// TwinCAT 3 PLC project ProgramPLC
// ProgramVersion: 3.1.4026.19
// libraries:
//   Tc2_DataExchange, * (Beckhoff Automation GmbH)
//   Tc2_Drive, * (Beckhoff Automation GmbH)
//   Tc2_EtherCAT, * (Beckhoff Automation GmbH)
//   Tc2_IoFunctions, * (Beckhoff Automation GmbH)
//   Tc2_Math, * (Beckhoff Automation GmbH)
//   Tc2_MC2, * (Beckhoff Automation GmbH)
//   Tc2_MC2_Camming, * (Beckhoff Automation GmbH)
//   Tc2_MC2_Drive, * (Beckhoff Automation GmbH)
//   Tc2_MC2_FlyingSaw, * (Beckhoff Automation GmbH)
//   Tc2_NC, * (Beckhoff Automation GmbH)
//   Tc2_Standard, * (Beckhoff Automation GmbH)
//   Tc2_SUPS, * (Beckhoff Automation GmbH)
//   Tc2_System, * (Beckhoff Automation GmbH)
//   Tc2_Utilities, * (Beckhoff Automation GmbH)
//   Tc3_EventLogger, * (Beckhoff Automation GmbH)
//   Tc3_Interfaces, * (Beckhoff Automation GmbH)
//   Tc3_IoLink, * (Beckhoff Automation GmbH)
//   Tc3_MC2_AdvancedHoming, * (Beckhoff Automation GmbH)
//   Tc3_Module, * (Beckhoff Automation GmbH)
//   Tc3_PackML, * (Beckhoff Automation GmbH)
//   TcEventLogger, * (Beckhoff Automation Poland)
//   Festo_VTEM_DevCon,3.5.7.235,Festo SE & Co. KG
// project tree:
//   DUTs/AxisControl/ ST_AxisControlHoldingBrake.TcDUT, ST_AxisControlLS.TcDUT, ST_AxisControlManual.TcDUT, ST_AxisControlManualHMI.TcDUT
//   DUTs/CapPreScrewer/ E_CapPreScrewer.TcDUT, ST_ADS_Read_Write.TcDUT, ST_ADS_Write.TcDUT, ST_CapPreScrewerCommandsIn.TcDUT, ST_CapPreScrewerParameters.TcDUT, ST_FormsCapSorter.TcDUT
//   DUTs/DUTsAdsCommunication/ ST_Communication.TcDUT, ST_MachinePermissions.TcDUT, ST_PackMLCmdForCom.TcDUT, ST_ReservedSignals.TcDUT
//   DUTs/DUTsAxisOnline/FBsIO/ ST_FBGetDriveRefIO.TcDUT, ST_FBHoldingBrakeCtrlIO.TcDUT, ST_FBMotorMonitoringIO.TcDUT, ST_FBNcSWLimitSwitchCtrlIO.TcDUT, ST_FBReadChannelErrorCodeIO.TcDUT, ST_FBSetPositionOffsetIO.TcDUT, ST_McAxisOnlineErrorCollection.TcDUT, ST_McAxisStatus.TcDUT, ST_MCHaltIO.TcDUT, ST_MCHomeIO.TcDUT, ST_MCJogIO.TcDUT, ST_MCMoveAbsoluteIO.TcDUT, ST_MCMoveModuloIO.TcDUT, ST_MCMoveRelativeIO.TcDUT, ST_MCMoveVelocityIO.TcDUT, ST_MCPowerIO.TcDUT, ST_MCReadDriveAddressIO.TcDUT, ST_MCReadParameterSetIO.TcDUT, ST_MCResetIO.TcDUT, ST_MCSetPositionIO.TcDUT, ST_MCStopIO.TcDUT
//   DUTs/DUTsAxisOnline/ ST_AX5000Diag.TcDUT, ST_McAxisOnline.TcDUT
//   DUTs/DUTsDiagnostics/ E_DiagState.TcDUT, ST_FrmWcDiag.TcDUT
//   DUTs/DUTsNew/ E_Actuator.TcDUT, E_Barrier.TcDUT, E_WeightLiftStationState.TcDUT
//   DUTs/DUTsPackMLStateMachine/ E_PackMLCommand.TcDUT, E_PackMLMode.TcDUT, E_PackMLState.TcDUT
//   DUTs/ E_BottleFeederState.TcDUT, E_CapFeederState.TcDUT, E_CapFeederState_1.TcDUT, E_CapPushingState.TcDUT, E_CatchStationState.TcDUT, E_CheckerState.TcDUT, E_ConveyorState.TcDUT, E_DispencerLifterState.TcDUT, E_DispencerState.TcDUT, E_DragStationState.TcDUT, E_DragStationStatePneum.TcDUT, E_EntranceGatesState.TcDUT, E_FestoEmcsStState.TcDUT, E_GripperScrewer.TcDUT, E_MachineState.TcDUT, E_MassHeatingState.TcDUT, E_PuckInserterState.TcDUT, E_RobotMovState.TcDUT, E_RollerScrewer.TcDUT, E_Station.TcDUT, E_WeightState.TcDUT, ST_MoverState.TcDUT, ST_Point.TcDUT, ST_Point_1.TcDUT, ST_SlotStatus.TcDUT, S_CycleTimes.TcDUT, S_Error.TcDUT, S_Information.TcDUT, S_PackageState.TcDUT, S_RFIDCheck.TcDUT, S_Warning.TcDUT
//   DUTs/ServerClientENUMS/ E_ConnectionSteps.TcDUT, E_ServerSteps.TcDUT
//   DUTs/Stations/LidFeeder/ E_LidFeederState.TcDUT
//   DUTs/Stations/LidSealer/ E_LidSealing.TcDUT
//   DUTs/Stations/WickFeeder/ E_WickFeederSorterState.TcDUT, E_WickFeederState.TcDUT
//   / GlobalTextList.TcGTLO, PlcTask.TcTTO, WeightTask.TcTTO
//   GVLs/ GVL.TcGVL, gvlChecks.TcGVL, gvlCommunication.TcGVL, GVL_CP.TcGVL, GVL_IO.TcGVL, GVL_ROPP.TcGVL, GVL_RS.TcGVL, Iterators.TcGVL, VIS.TcGVL, VIS_CP.TcGVL, VIS_M.TcGVL, VIS_RFID.TcGVL, VIS_ROPP.TcGVL, VIS_RS.TcGVL
//   GVLs/UVFF/ GVL_Recipe.TcGVL, GVL_UVFF.TcGVL, GVL_VIS.TcGVL
//   POUs/FB/ADSCommumication/ FB_AdsCommunicationRead.TcPOU
//   POUs/FB/AxisControl/AX8000/ FB_AxisAX8000.TcPOU, I_AxisControlPhysical.TcIO
//   POUs/FB/AxisControl/Base/ FB_AxisBase.TcPOU, I_AxisControlBase.TcIO
//   POUs/FB/AxisControl/Internal/ FB_FilterEx_2.TcPOU, FB_GetDriveRef_1.TcPOU, FB_HoldingBrakeCtrlAX8000_1.TcPOU, FB_NcPosLagMonitoring.TcPOU, FB_NcSWLimitSwitchCtrlv2.TcPOU, FB_ReadChannelErrorCodeAX8000_1.TcPOU, F_AX8xErrMsg_2.TcPOU, F_AxErrMsg_2.TcPOU
//   POUs/FB/AxisControl/Internal/HomingAdv/ FB_HomingLimitSwitch.TcPOU, FB_HomingMemoryAX8000.TcPOU, FB_HomingTorqueDetection.TcPOU, FB_HomingTorqueDetectionSensor.TcPOU, FB_HomingTorque_1.TcPOU
//   POUs/FB/Axis/ F_AX8xErrMsg.TcPOU, F_AxErrMsg.TcPOU
//   POUs/FB/Blinkers/ FB_Blink_AS.TcPOU, FB_Blink_S.TcPOU, FUN_Beep.TcPOU
//   POUs/FB/Charts/ FB_ChartGenerator.TcPOU, FB_SimplePulseGenerator.TcPOU, FB_WeightHistory.TcPOU
//   POUs/FB/Conversions/ ArrayOfReal_To_String.TcPOU, arrBOOL16_TO_WORD.TcPOU, arrBOOL8_TO_BYTE.TcPOU, ArrOfInt_To_String.TcPOU, FB_CONCAT_S2040.TcPOU, FB_DIntTo4Byte.TcPOU, FB_IntTo2Byte.TcPOU, F_4BYTES_TO_DWORD.TcPOU, F_4BYTES_TO_REAL.TcPOU, F_8BYTES_TO_LREAL.TcPOU, F_BCDToDec.TcPOU, F_CLEAN_S2040.TcPOU, F_Convert_4BBCD_To_Real.TcPOU, F_DWORD_TO_REAL.TcPOU, F_Words_to_Real.TcPOU, GRAYB_TO_WORD.TcPOU, GRAYW_TO_WORD.TcPOU
//   POUs/FB/Conversions/BitOriented/ BCD_TO_INT.TcPOU, F_1stByteW.TcPOU, F_1stByteWtoB.TcPOU, F_2Bytes_To_Word.TcPOU, F_2ndByteW.TcPOU, F_2ndByteWtoB.TcPOU, F_MaskWord.TcPOU, L_TBConvArrBitsToDword.TcPOU, L_TBConvBitsToByte.TcPOU, L_TBConvBitsToDword.TcPOU, L_TBConvBitsToWord.TcPOU, L_TBConvByteToBits.TcPOU, L_TBConvDwordToArrBits.TcPOU, L_TBConvDwordToBits.TcPOU, L_TBConvWordToBits.TcPOU, L_TBGetBitOfByte.TcPOU, L_TBGetBitOfDword.TcPOU, L_TBGetBitOfWord.TcPOU, L_TBResetBitOfByte.TcPOU, L_TBResetBitOfDword.TcPOU, L_TBResetBitOfWord.TcPOU, L_TBSetBitOfByte.TcPOU, L_TBSetBitOfDword.TcPOU, L_TBSetBitOfWord.TcPOU, L_TBSquareWave.TcPOU
//   POUs/FB/DateAndTime/ FB_GetSystemTime.TcPOU, FB_SimpleWorkTime.TcPOU, FB_TimeMeasureEx.TcPOU, FB_WorktimeCompact.TcPOU
//   POUs/FB/Diagnostics/FBsDiagnostic/ FB_AdvancedLogEvent.TcPOU, FB_AntiBlinkAlarmFilter.TcPOU, FB_TaskInfo.TcPOU
//   POUs/FB/Diagnostics/POUsDiagnosticComponents/Checks/ CheckBounds.TcPOU, CheckDivDInt.TcPOU, CheckDivLInt.TcPOU, CheckDivLReal.TcPOU, CheckDivReal.TcPOU, CheckPointer.TcPOU, CheckRangeSigned.TcPOU, CheckRangeUnsigned.TcPOU, P_Checks.TcPOU
//   POUs/FB/Diagnostics/POUsDiagnosticComponents/ P_EtherCAT_ChangeCounter.TcPOU, P_EtherCAT_Diag.TcPOU, P_GroupsWcStates.TcPOU, P_Persistent.TcPOU, P_PlcTaskSystemInfo.TcPOU, P_SystemDiag_EventLog.TcPOU, P_SystemInfo.TcPOU, P_TaskInfo.TcPOU
//   POUs/FB/ FB_2GripperScrewers.TcPOU, FB_2GripperScrewers_New.TcPOU, FB_2ReasonBadPackageWithID.TcPOU, FB_BalluffBMP0005.TcPOU, FB_BeckhoffEL3356Weight.TcPOU, FB_CapFeeder.TcPOU, FB_CapPreScrewer.TcPOU, FB_CapPusher.TcPOU, FB_CapPusherFeeder.TcPOU, FB_DigitalInput_1.TcPOU, FB_Robot2Bottles.TcPOU, FB_CapFeeder_old.TcPOU, FB_CatchStation.TcPOU, FB_CatchStationEnkoder.TcPOU, FB_CatchStationEnkoder_old.TcPOU (excluded from build), FB_Checker.TcPOU, FB_CycleTimes.TcPOU, FB_EntranceGatesServo.TcPOU, FB_FestoEmcsSt.TcPOU, FB_HomingTorque.TcPOU, FB_IfmIoLinkRfid.TcPOU, FB_InputFilter.TcPOU, FB_JiesangActuatorEncoder.TcPOU, FB_JiesangActuatorEncoder_1.TcPOU, FB_JiesangActuatorEncoderModul.TcPOU, FB_LenzeInverter.TcPOU, FB_LidFeeder.TcPOU, FB_LidSealer.TcPOU, FB_MitsubishiInverter.TcPOU, FB_MoveRegister.TcPOU, FB_MoveRegister4.TcPOU, FB_MoveRegisterCapControl.TcPOU, FB_MoveRegisterROPPCapControl.TcPOU, FB_MoveRegisterSortAndMove.TcPOU, FB_MoveRegisterSortAndMoveLF.TcPOU, FB_MoveRegisterLF.TcPOU, FB_MoveRegisterSortAndMoveROPP.TcPOU, FB_OEECycleTimes.TcPOU, FB_OEERejectionReason.TcPOU, FB_ReasonBadPackage.TcPOU, FB_RollerScrewer.TcPOU, FB_ROPPCapping.TcPOU, FB_ROPPFeeder.TcPOU, FB_SensorDiag.TcPOU, FB_ServoDispencerServoLifter.TcPOU, FB_ServoDispencerServoLifter_kopia_przed_akt_XTS.TcPOU, FB_SpringGateV2.TcPOU, FB_State.TcPOU, FB_TankHeating.TcPOU, FB_TempRegulator.TcPOU, FB_VisionChecker.TcPOU, FB_VisionChecker_new.TcPOU, FB_WeightCorrection.TcPOU, FB_WickFeederStation.TcPOU, FB_WriteDataToArrayOfArrays.TcPOU, FB_WriteDataToArrayString.TcPOU, FB_WriteRFID.TcPOU, FB_WriteRFIDnew.TcPOU, FB_AutoTrialRenew_ADS.TcPOU, F_StringToWstringPL.TcPOU, FB_InputFilter_v2.TcPOU
//   POUs/FB/FileAccess/ FB_ReadTextFromFile.TcPOU, FB_SaveTextToFile.TcPOU, FB_FileLog.TcPOU, FB_SaveLineToFile.TcPOU
//   POUs/FB/Led/ FB_PackMlToRgb_EL2564.TcPOU, FB_RgbLedTape_EL2563.TcPOU
//   POUs/FB/NC/ FB_PWM_BASIC.TcPOU
//   POUs/FB/NewFBs/ FB_BottleFeeder.TcPOU, FB_CatchStationWithSensor.TcPOU, FB_FormsDragStepper.TcPOU, FB_FormsDragActuator.TcPOU, FB_Gate.TcPOU, FB_PucksInserter.TcPOU, FB_SensorAcetone.TcPOU, FB_SensorFlow.TcPOU, FB_WeightStation.TcPOU
//   POUs/FB/POUsAxisOnline/AX5000/ FB_AxisDiag.TcPOU, FB_ChangeEtherCATSlaveState.TcPOU, FB_HoldingBrakeCtrlAX5000.TcPOU, FB_McAxisOnlineAX5000.TcPOU, FB_MotorMonitoringAX5000.TcPOU, FB_SetPositionOffset.TcPOU, F_AX5xErrMsg.TcPOU
//   POUs/FB/POUsAxisOnline/AX8000/ FB_HoldingBrakeCtrlAX8000.TcPOU, FB_McAxisOnlineAX8000.TcPOU, FB_MotorMonitoringAX8000.TcPOU, FB_ReadChannelErrorCodeAX8000.TcPOU, F_AX8xErrMsg_1.TcPOU
//   POUs/FB/POUsAxisOnline/EL72xx/ FB_HoldingBrakeCtrlEL72xx.TcPOU, FB_McAxisOnlineEL72xx.TcPOU, FB_MotorMonitoringEL72xx.TcPOU, FB_ReadChannelErrorCodeEL72xx.TcPOU, F_EL72ErrMsg.TcPOU
//   POUs/FB/POUsAxisOnline/FBs/ FB_FilterEx_1.TcPOU, FB_GetDriveRef.TcPOU, FB_NcSWLimitSwitchCtrl.TcPOU, F_AxErrMsg_1.TcPOU
//   POUs/FB/POUsAxisOnline/NC/ FB_McAxisOnlineNC.TcPOU
//   POUs/FB/Various/ FB_4_20mA_TO_INT.TcPOU, FB_Average.TcPOU, FB_FilterEx.TcPOU, FB_Persistent.TcPOU, FB_PIDBasic.TcPOU, FB_Skalowanie.TcPOU, F_ScaleLREAL.TcPOU, F_Scaling.TcPOU
//   POUs/ MAIN.TcPOU, P00_Alarms.TcPOU, P00_Basic.TcPOU, P00_Counters.TcPOU, P00_OEE.TcPOU, P00_Persistent.TcPOU, P00_Communication.TcPOU, P00_PneumaticValves.TcPOU, P00_ReadRFIDCard.TcPOU, P00_Recipes.TcPOU, P00_SensorDiagnostics.TcPOU, P00_Signalization.TcPOU, P00_SystemDiagnostics.TcPOU, P00_Visualization.TcPOU, P01_BottleFeeder.TcPOU, P00_PackML.TcPOU, P01_BottleSorter.TcPOU, P01_PucksInserter.TcPOU, P01_TwoPhasesBarriers.TcPOU, P02_BottlePusher.TcPOU, P02_Dispencers.TcPOU, P05_Weight.TcPOU, P06_WickFeeder.TcPOU, P07_CapPusher.TcPOU, P07_ROPP.TcPOU, P08_CapFeeder.TcPOU, P01_Gates.TcPOU, P05_WeightCorrection.TcPOU, P06_LidFeeder.TcPOU, P06_LidPuttedCheck.TcPOU, P06_LidSealer.TcPOU, P08_CapSorter.TcPOU, P09_CapPuttedCheck.TcPOU, P10_GripperScrewer.TcPOU, P11_CapCorrectCheck.TcPOU, P11_RollerScrewer.TcPOU, P13_BottleTransferAfterDrag.TcPOU, P13_BottleTransfer.TcPOU, P14_BadBottleConyevor.TcPOU, P15_FormTransporters.TcPOU, P16_LabelMachine.TcPOU, P17_TurnTables.TcPOU, P02_DispencersCharts.TcPOU, P200_CapPreScrewer.TcPOU, P20_ExhaustFan.TcPOU, P20_ExhaustFan_old.TcPOU, P_AdsLicenseServer.TcPOU, P_WenglorTeach.TcPOU
//   POUs/Recipes/NewRecipes/Components/ ST_BoolParametr.TcDUT, ST_DiParametrr.TcDUT, ST_LrParametr.TcDUT, ST_TextListParametr.TcDUT, ST_UdiParametr.TcDUT
//   POUs/Recipes/NewRecipes/ E_MacroProductProcessRegister.TcDUT, E_ProductType.TcDUT, ST_Recipe.TcDUT, ST_RecipeListItem.TcDUT, ST_Recipe_UBF_PARAM.TcDUT, ST_Recipe_UBL_PARAM.TcDUT, ST_Recipe_UCF_PARAM.TcDUT
//   POUs/Recipes/NewRecipes/RecipeCSV/ FB_ListSaveCSV.TcPOU, FB_LoadCSV.TcPOU, FB_RecipeSaveCSV.TcPOU, FB_RecipeVariablesSaveCSV.TcPOU
//   POUs/Recipes/NewRecipes/RecipeList/ E_FileOpSteps.TcDUT, FB_Load.TcPOU, FB_Save.TcPOU
//   POUs/Recipes/NewRecipes/RecipeParts/ ST_BoxRobotRecipe.TcDUT, ST_DownTransporterRecipe.TcDUT, ST_DymmyStationRecipe.TcDUT, ST_ExtMachineRecipe.TcDUT, ST_InBoxControlRecipe.TcDUT, ST_InTransporterRecipe.TcDUT, ST_LeftRightCloserValveRecipe.TcDUT, ST_LiftedTableRecipe.TcDUT, ST_LRTransporterRecipe.TcDUT, ST_MacroBoxFeedingProcessRecipe.TcDUT, ST_MacroBoxingProcessRecipe.TcDUT, ST_MacroInProcessRecipe.TcDUT, ST_MacroMachineProcessRecipe.TcDUT, ST_MacroProductProcessRecipe.TcDUT, ST_MacroTransportRecipe.TcDUT, ST_MainProcessRecipe.TcDUT, ST_MainSystemRecipe.TcDUT, ST_MoverPressValveRecipe.TcDUT, ST_OutControlRecipe.TcDUT, ST_ProductBoxerRecipe.TcDUT, ST_ProductRobotRecipe.TcDUT, ST_ProductTableCoverRecipe.TcDUT, ST_RejectBuforRecipe.TcDUT, ST_SpareElementsLockRecipe.TcDUT, ST_StandartGateRecipe.TcDUT, ST_StepMoverRecipe.TcDUT
//   POUs/Recipes/ P009_ReadSavePersistent.TcPOU, P010_AlarmsWarningsInfosLogs.TcPOU, P020_RtcEffectivityOEE.TcPOU, P030_Recipes.TcPOU
// real-time tasks:
//   TASK MainTask: cycle T#3ms, priority 20, ADS port 350
//   TASK SafetyTask: cycle T#10ms, priority 22, ADS port 351
//   TASK WeightTask: cycle T#2ms, priority 19, ADS port 354
//   TASK PlcTask: cycle T#10ms, priority 21, ADS port 355
//   TASK TaskToRefreshEAP: cycle T#1ms, priority 12, ADS port 301
// motion (NC):
//   TASK NC-Task 1 SAF: cycle T#2ms, priority 4, ADS port 501
//   TASK NC-Task 1 SVB: cycle T#10ms, priority 8, ADS port 511
//   AXIS Doz1 (id 1)
//   AXIS Doz2 (id 2)
//   AXIS Doz3 (id 3)
//   AXIS Doz4 (id 4)
//   AXIS PodDoz12 (id 5)
//   AXIS PodDoz34 (id 6)
//   AXIS Zak1 (id 7)
//   AXIS PodZak1 (id 8)
//   AXIS Zak2 (id 9)
//   AXIS PodZak2 (id 10)
//   AXIS PrzecDoz (id 11)
//   AXIS PrzecDoz2 (id 12)
//   AXIS PrzecZak (id 13)
//   AXIS PrzecSorNak (id 14)
//   AXIS PrzecPlat (id 15)
//   AXIS PrzecGrz (id 16)
//   AXIS VirtualDos (id 17)
//   AXIS VirtualPodDoz (id 18)
//   AXIS ZakEncoder1 (id 19)
//   AXIS ZakEncoder2 (id 20)
//   AXIS PI_Karusela (id 21)
//     General: UnitName=Degree, UnitFlags=#x00000004
//     Dynamic: Acceleration=15000, Deceleration=15000, Jerk=225000
//     OtherSettings: AllowMotionCmdToSlave=true
//     encoder EncType=19
//       EncPara: ScaleFactorDenominator=8, ToleranceWndModuloStart=1, Inverse=true, MaxCount=#x0036ee80, ReferenceSystem=2
//         Inc: RefSoftSyncMask=#x0036ee80
//         TimeComp: TimeCompMode=1, EncDelayCycles=4
//     drive DrvType=16
//       DrvPara: Inverse=true, MaxCount=#xffffffff, DriveControlDWord=#x00020000
//         Analog: TorqueSetpointScale=10, ScaleFactorActTorque=0.1
//         TimeComp: TimeCompMode=1, TaskDelayCycles=1
//     controller CtrType=1
//       CtrPara: PriorControlFactor=1
//         PosDiffControl: Enable=false
//         Observer: BandWidth=20
//   AXIS RC40_Zak1 (id 22)
//     General: UnitName=°
//     Dynamic: Acceleration=15000, Deceleration=15000, Jerk=71262.9405
//     Velo: RefSearch=158.36209, RefSync=158.36209, SlowManual=791.81045, FastManual=4750.8627, Fast=15836.209, Maximum=15836.209
//     OtherSettings: AllowMotionCmdToSlave=true
//     encoder EncType=8
//       EncPara: ScaleFactorNumerator=70920, ScaleFactorDenominator=262144000, MaxCount=#xffffffff, EncPositionSource=1
//     drive DrvType=9
//       DrvPara: MaxCount=#xffffffff, DriveControlDWord=#x00030100
//         Analog: VeloReferenz=17419.8299, VeloScale=1.02400649589962, TorqueSetpointScale=10, ScaleFactorActTorque=0.1
//         TimeComp: TaskDelayCycles=1
//     controller CtrType=1
//       CtrPara: PriorControlFactor=1
//         Observer: BandWidth=20
//   AXIS RC40_Zak2 (id 23)
//     General: UnitName=°
//     Dynamic: Acceleration=15000, Deceleration=15000, Jerk=71262.9405
//     Velo: RefSearch=158.36209, RefSync=158.36209, SlowManual=791.81045, FastManual=4750.8627, Fast=15836.209, Maximum=15836.209
//     OtherSettings: AllowMotionCmdToSlave=true
//     encoder EncType=8
//       EncPara: ScaleFactorNumerator=70920, ScaleFactorDenominator=262144000, MaxCount=#xffffffff
//     drive DrvType=9
//       DrvPara: MaxCount=#xffffffff, DriveControlDWord=#x00030100
//         Analog: VeloReferenz=17419.8299, VeloScale=1.02400649589962, TorqueSetpointScale=10, ScaleFactorActTorque=0.1
//         TimeComp: TaskDelayCycles=1
//     controller CtrType=1
//       CtrPara: PriorControlFactor=1
//         Observer: BandWidth=20
//   AXIS UVFF_Zak (id 24)
//     General: UnitName=°
//     Dynamic: AccelerationMaximum=100000, DecelerationMaximum=100000, Acceleration=12554.4, Deceleration=12554.4, Jerk=37663.3
//     Velo: RefSearch=83.69612, RefSync=83.69612, SlowManual=10, FastManual=250, Fast=8369.612, Maximum=8369.61
//     PositionAreaControl: Enable=false
//     TargetPosControl: Enable=false
//     OtherSettings: AllowMotionCmdToSlave=true
//     encoder EncType=19
//       EncPara: ScaleFactorNumerator=360, ScaleFactorDenominator=4294967296, Inverse=true, EncMode=3, MaxCount=#xffffffff
//         FilterTime: TVelo=0, TAcc=0
//         Inc: RefSoftSyncMask=#x6aaaaaaa
//         TimeComp: TimeCompMode=1, EncDelayCycles=1
//     drive DrvType=16
//       DrvPara: Inverse=true, MaxCount=#xffffffff, DriveControlDWord=#x00020100
//         Analog: VeloReferenz=9206.5732, VeloScale=71.5255737304688, TorqueSetpointScale=10, ScaleFactorActTorque=0.1
//         TimeComp: TaskDelayCycles=1, AdditionalTimeShift=6000
//     controller CtrType=1
//       CtrPara: PriorControlFactor=1
//         PosDiffControl: Enable=false, Range=600
//         Observer: BandWidth=20
//   AXIS UVFF_Os_Y (id 25)
//     Dynamic: Acceleration=10000, Deceleration=10000, Jerk=50000.3
//     Velo: RefSearch=14.33405, RefSync=14.33405, SlowManual=4, FastManual=30, Fast=1433.405, Maximum=1433.4
//     OtherSettings: AllowMotionCmdToSlave=true
//     encoder EncType=19
//       EncPara: ScaleFactorNumerator=125, ScaleFactorDenominator=5242880, MaxCount=#xffffffff
//         SoftEndMinControl: Range=-30
//         SoftEndMaxControl: Enable=true, Range=550
//     drive DrvType=16
//       DrvPara: MaxCount=#xffffffff, DriveControlDWord=#x00020100
//         Analog: VeloReferenz=1576.7455, TorqueSetpointScale=10, ScaleFactorActTorque=0.1
//         TimeComp: TaskDelayCycles=1
//     controller CtrType=1
//       CtrPara: PriorControlFactor=1
//         PosDiffControl: Range=10
//         Observer: BandWidth=20
//   AXIS UVFF_Os_Z (id 26)
//     Dynamic: AccelerationMaximum=30000, DecelerationMaximum=30000, Acceleration=10000, Deceleration=10000, Jerk=50000
//     Velo: RefSearch=35.01545, RefSync=35.01545, SlowManual=4, FastManual=40, Fast=3501.545, Maximum=3501.55
//     OtherSettings: AllowMotionCmdToSlave=true
//     encoder EncType=19
//       EncPara: ScaleFactorNumerator=96, ScaleFactorDenominator=3145728, MaxCount=#xffffffff
//         SoftEndMaxControl: Enable=true, Range=451
//     drive DrvType=16
//       DrvPara: MaxCount=#xffffffff, DriveControlDWord=#x00020100
//         Analog: VeloReferenz=3851.6995, TorqueSetpointScale=10, ScaleFactorActTorque=0.1
//         TimeComp: TaskDelayCycles=1
//     controller CtrType=1
//       CtrPara: PriorControlFactor=1
//         Observer: BandWidth=20
//   AXIS UVFF_VirtualAxis (id 27)
//     Dynamic: AccelerationMaximum=1500000000, DecelerationMaximum=1500000000, Acceleration=1500000000, Deceleration=1500000000, Jerk=10000000000
//     Velo: SlowManual=10, Maximum=3501.55
//     PositionAreaControl: Enable=false
//     TargetPosControl: Enable=false
//     OtherSettings: AllowMotionCmdToSlave=true
//     encoder EncType=1
//     drive DrvType=5
//       Analog: VeloReferenz=3851.6995, TorqueSetpointScale=10, ScaleFactorActTorque=0.1
//       TimeComp: TaskDelayCycles=1
//     controller CtrType=1
//       CtrPara: PriorControlFactor=1
//         PosDiffControl: Enable=false
//         Observer: BandWidth=20
// I/O:
//   DEVICE Device 1 (EtherCAT)
//   DEVICE Device 2 (EtherCAT Automation Protocol), AmsNetId 0.0.0.0.2.1
//     UF50 Publisher
//     UF50  Subscriber
//     UP50B Publisher
//     UP50B  Subscriber
// variable links:
//   Device 1 (EtherCAT) <-> Device 2 (EtherCAT Automation Protocol)/UF50  Subscriber
//     R2_BC1 (EK1100)/CO2 (EL6910)/ConnectionOutputs/TwinSafeGroup3.EL6910_CommModule_151 RxPDO <-> Sub-Var 1/Inputs/VarData
//   Device 1 (EtherCAT) <-> Device 2 (EtherCAT Automation Protocol)/UF50 Publisher
//     R2_BC1 (EK1100)/CO2 (EL6910)/ConnectionInputs/TwinSafeGroup3.EL6910_CommModule_151 TxPDO <-> Pub-Var 1/Outputs/VarData
//   Device 1 (EtherCAT) <-> Device 2 (EtherCAT Automation Protocol)/UP50B  Subscriber
//     R2_BC1 (EK1100)/CO2 (EL6910)/ConnectionOutputs/TwinSafeGroup2.EL6910_CommModule_152 RxPDO <-> Sub-Var 1/Inputs/VarData
//   Device 1 (EtherCAT) <-> Device 2 (EtherCAT Automation Protocol)/UP50B Publisher
//     R2_BC1 (EK1100)/CO2 (EL6910)/ConnectionInputs/TwinSafeGroup2.EL6910_CommModule_152 TxPDO <-> Pub-Var 1/Outputs/VarData
//   TaskToRefreshEAP <-> Device 2 (EtherCAT Automation Protocol)
//     Inputs/EAP_State <-> Inputs/DevState
//   Axes/PI_Karusela <-> Device 1 (EtherCAT)/R2_242A1 (CU1128)/R2_242A1 (CU1128-C)/PI_71U1 (ctrlX DRIVE XCS (CoE))
//     Drive/Inputs/In/nDcOutputTime <-> InfoData/DcOutputShift
//     Drive/Inputs/In/nState1 <-> Module 1 (Cyclic Sync Postion Mode)/Transmit PDO Mapping Parameter/CiA 402 status word
//     Drive/Inputs/In/nState2 <-> Module 1 (Cyclic Sync Postion Mode)/Transmit PDO Mapping Parameter/CiA 402 status word @bit 8
//     Drive/Inputs/In/nState4 @bit 1 <-> WcState/InputToggle
//     Drive/Inputs/In/nState4 <-> WcState/WcState
//     Drive/Outputs/Out/nCtrl1 <-> Module 1 (Cyclic Sync Postion Mode)/Receive PDO Mapping Parameter/CiA 402 control word
//     Drive/Outputs/Out/nCtrl2 <-> Module 1 (Cyclic Sync Postion Mode)/Receive PDO Mapping Parameter/CiA 402 control word @bit 8
//     Drive/Outputs/Out/nDataOut1 <-> Module 1 (Cyclic Sync Postion Mode)/Receive PDO Mapping Parameter/Target position
//     Enc/Inputs/In/nDataIn1 <-> Module 1 (Cyclic Sync Postion Mode)/Transmit PDO Mapping Parameter/Position actual value
//     Enc/Inputs/In/nDcInputTime <-> InfoData/DcInputShift
//     Enc/Inputs/In/nState4 @bit 1 <-> WcState/InputToggle
//     Enc/Inputs/In/nState4 <-> WcState/WcState
//   Axes/RC40_Zak1 <-> Device 1 (EtherCAT)/R2_242A1 (CU1128)/R2_242A1 (CU1128-B)/RC40_ZAK_1_2 (AX5203-0000-0213)
//     Drive/Inputs/In/nDataIn1 <-> AT 1/Following distance
//     Drive/Inputs/In/nDataIn3[0] <-> AT 1/Torque/force feedback value
//     Drive/Inputs/In/nDcOutputTime <-> InfoData/DcOutputShift
//     Drive/Inputs/In/nState1 <-> AT 1/Drive status word @bit 8
//     Drive/Inputs/In/nState2 <-> AT 1/Drive status word
//     Drive/Inputs/In/nState4 @bit 1 <-> WcState/InputToggle
//     Drive/Inputs/In/nState4 <-> WcState/WcState
//     Drive/Outputs/Out/nCtrl1 <-> MDT 1/Master control word @bit 8
//     Drive/Outputs/Out/nDataOut1 <-> MDT 1/Position command value
//     Enc/Inputs/In/nDataIn1 <-> AT 1/Position feedback 1 value
//     Enc/Inputs/In/nDcInputTime <-> InfoData/DcInputShift
//     Enc/Inputs/In/nState4 @bit 1 <-> WcState/InputToggle
//     Enc/Inputs/In/nState4 <-> WcState/WcState
//   Axes/RC40_Zak2 <-> Device 1 (EtherCAT)/R2_242A1 (CU1128)/R2_242A1 (CU1128-B)/RC40_ZAK_1_2 (AX5203-0000-0213)
//     Drive/Inputs/In/nDataIn1 <-> AT 2/Following distance
//     Drive/Inputs/In/nDataIn3[0] <-> AT 2/Torque/force feedback value
//     Drive/Inputs/In/nDcOutputTime <-> InfoData/DcOutputShift
//     Drive/Inputs/In/nState1 <-> AT 2/Drive status word @bit 8
//     Drive/Inputs/In/nState2 <-> AT 2/Drive status word
//     Drive/Inputs/In/nState4 @bit 1 <-> WcState/InputToggle
//     Drive/Inputs/In/nState4 <-> WcState/WcState
//     Drive/Outputs/Out/nCtrl1 <-> MDT 2/Master control word @bit 8
//     Drive/Outputs/Out/nDataOut1 <-> MDT 2/Position command value
//     Enc/Inputs/In/nDataIn1 <-> AT 2/Position feedback 1 value
//     Enc/Inputs/In/nDcInputTime <-> InfoData/DcInputShift
//     Enc/Inputs/In/nState4 @bit 1 <-> WcState/InputToggle
//     Enc/Inputs/In/nState4 <-> WcState/WcState
//   (this object) <-> Device 1 (EtherCAT)
//     PlcTask Inputs/P_EtherCAT_Diag.uiDevState <-> Inputs/DevState
//     PlcTask Inputs/P_EtherCAT_Diag.uiFrmWcState[1] <-> Inputs/Frm0State
//   (this object) <-> Device 1 (EtherCAT)/600U1 (AX8620-0000-0105)/604U1_Zak1Pod1 (AX8206-0100-0106)
//     PlcTask Outputs/P10_GripperScrewer.QnGripperScrewer1ProportionalGain <-> Ch A/Ch A PositionControl Outputs/Position control proportional gain
//     PlcTask Outputs/P10_GripperScrewer.QnGripperScrewer1TorqueLimit <-> Ch A/Ch A TorqueControl Outputs/Ch A Bipolar torque/force limit value
//   (this object) <-> Device 1 (EtherCAT)/600U1 (AX8620-0000-0105)/605U1_Zak2Pod2 (AX8206-0100-0106)
//     PlcTask Outputs/P10_GripperScrewer.QnGripperScrewer2ProportionalGain <-> Ch A/Ch A PositionControl Outputs/Position control proportional gain
//     PlcTask Outputs/P10_GripperScrewer.QnGripperScrewer2TorqueLimit <-> Ch A/Ch A TorqueControl Outputs/Ch A Bipolar torque/force limit value
//   (this object) <-> Device 1 (EtherCAT)/R1_615U1_Knoty (FR-E800-E)
//     PlcTask Inputs/P06_WickFeeder.InWickFeederSorterSTW <-> 1st Transmit PDO Mapping/Statusword
//     PlcTask Inputs/P06_WickFeeder.InWickFeederSorterVelocityCV <-> 1st Transmit PDO Mapping/Index:Pr.1330,Sub:Pr.1394(Low)
//     PlcTask Outputs/P06_WickFeeder.QnWickFeederSorterCTW <-> 1st Receive PDO Mapping/Controlword
//     PlcTask Outputs/P06_WickFeeder.QnWickFeederSorterVelocitySV <-> 1st Receive PDO Mapping/Index:Pr.1320,Sub:Pr.1389(Low)
//   (this object) <-> Device 1 (EtherCAT)/R2_242A1 (CU1128)/R1_610U1_PI-Doz (FR-E800-E)
//     PlcTask Inputs/P15_FormTransporters.InFormTransporterDispencerSTW <-> 1st Transmit PDO Mapping/Statusword
//     PlcTask Inputs/P15_FormTransporters.InFormTransporterDispencerVelocityCV <-> 1st Transmit PDO Mapping/Index:Pr.1330,Sub:Pr.1394(Low)
//     PlcTask Outputs/P15_FormTransporters.QnFormTransporterDispencerCTW <-> 1st Receive PDO Mapping/Controlword
//     PlcTask Outputs/P15_FormTransporters.QnFormTransporterDispencerVelocitySV <-> 1st Receive PDO Mapping/Index:Pr.1320,Sub:Pr.1389(Low)
//   (this object) <-> Device 1 (EtherCAT)/R2_242A1 (CU1128)/R1_611U1_Doz-Nakr (FR-E800-E)
//     PlcTask Inputs/P15_FormTransporters.InFormTransporterScrewerSTW <-> 1st Transmit PDO Mapping/Statusword
//     PlcTask Inputs/P15_FormTransporters.InFormTransporterScrewerVelocityCV <-> 1st Transmit PDO Mapping/Index:Pr.1330,Sub:Pr.1394(Low)
//     PlcTask Outputs/P15_FormTransporters.QnFormTransporterScrewerCTW <-> 1st Receive PDO Mapping/Controlword
//     PlcTask Outputs/P15_FormTransporters.QnFormTransporterScrewerVelocitySV <-> 1st Receive PDO Mapping/Index:Pr.1320,Sub:Pr.1389(Low)
//   (this object) <-> Device 1 (EtherCAT)/R2_242A1 (CU1128)/R1_612U1_Nakr-BufZakr (FR-E800-E)
//     PlcTask Inputs/P15_FormTransporters.InFormTransporterAfterCapSorterSTW <-> 1st Transmit PDO Mapping/Statusword
//     PlcTask Inputs/P15_FormTransporters.InFormTransporterAfterCapSorterVelocityCV <-> 1st Transmit PDO Mapping/Index:Pr.1330,Sub:Pr.1394(Low)
//     PlcTask Outputs/P15_FormTransporters.QnFormTransporterAfterCapSorterCTW <-> 1st Receive PDO Mapping/Controlword
//     PlcTask Outputs/P15_FormTransporters.QnFormTransporterAfterCapSorterVelocitySV <-> 1st Receive PDO Mapping/Index:Pr.1320,Sub:Pr.1389(Low)
//   (this object) <-> Device 1 (EtherCAT)/R2_242A1 (CU1128)/R1_613U1_BufZak-Zakr (FR-E800-E)
//     PlcTask Inputs/P15_FormTransporters.InFormTransporterBeforeScrewerSTW <-> 1st Transmit PDO Mapping/Statusword
//     PlcTask Inputs/P15_FormTransporters.InFormTransporterBeforeScrewerVelocityCV <-> 1st Transmit PDO Mapping/Index:Pr.1330,Sub:Pr.1394(Low)
//     PlcTask Outputs/P15_FormTransporters.QnFormTransporterBeforeScrewerCTW <-> 1st Receive PDO Mapping/Controlword
//     PlcTask Outputs/P15_FormTransporters.QnFormTransporterBeforeScrewerVelocitySV <-> 1st Receive PDO Mapping/Index:Pr.1320,Sub:Pr.1389(Low)
//   (this object) <-> Device 1 (EtherCAT)/R2_242A1 (CU1128)/R1_614U1_Zakr-Robot (FR-E800-E)
//     PlcTask Inputs/P15_FormTransporters.InFormTransporterAfterScrewerSTW <-> 1st Transmit PDO Mapping/Statusword
//     PlcTask Inputs/P15_FormTransporters.InFormTransporterAfterScrewerVelocityCV <-> 1st Transmit PDO Mapping/Index:Pr.1330,Sub:Pr.1394(Low)
//     PlcTask Outputs/P15_FormTransporters.QnFormTransporterAfterScrewerCTW <-> 1st Receive PDO Mapping/Controlword
//     PlcTask Outputs/P15_FormTransporters.QnFormTransporterAfterScrewerVelocitySV <-> 1st Receive PDO Mapping/Index:Pr.1320,Sub:Pr.1389(Low)
//   (this object) <-> Device 1 (EtherCAT)/R2_242A1 (CU1128)/R1_630U1 (Anybus CompactCom 40 EtherCAT)
//     PlcTask Inputs/P13_BottleTransfer.IaDataRobotIO[1] <-> Transmit PDO Mapping/SubIndex 001
//     PlcTask Inputs/P13_BottleTransfer.IaDataRobotIO[2] <-> Transmit PDO Mapping/SubIndex 002
//     PlcTask Inputs/P13_BottleTransfer.IaDataRobotIO[3] <-> Transmit PDO Mapping/SubIndex 003
//     PlcTask Inputs/P13_BottleTransfer.IaDataRobotIO[4] <-> Transmit PDO Mapping/SubIndex 004
//     PlcTask Inputs/P13_BottleTransfer.IaDataRobotIO[5] <-> Transmit PDO Mapping/SubIndex 005
//     PlcTask Inputs/P13_BottleTransfer.IaDataRobotIO[6] <-> Transmit PDO Mapping/SubIndex 006
//     PlcTask Inputs/P13_BottleTransfer.IaDataRobotIO[7] <-> Transmit PDO Mapping/SubIndex 007
//     PlcTask Inputs/P13_BottleTransfer.IaDataRobotIO[8] <-> Transmit PDO Mapping/SubIndex 008
//     PlcTask Inputs/P13_BottleTransfer.IaDataRobotREG[10] <-> Transmit PDO Mapping/SubIndex 010
//     PlcTask Inputs/P13_BottleTransfer.IaDataRobotREG[11] <-> Transmit PDO Mapping/SubIndex 011
//     PlcTask Inputs/P13_BottleTransfer.IaDataRobotREG[12] <-> Transmit PDO Mapping/SubIndex 012
//     PlcTask Inputs/P13_BottleTransfer.IaDataRobotREG[13] <-> Transmit PDO Mapping/SubIndex 013
//     PlcTask Inputs/P13_BottleTransfer.IaDataRobotREG[14] <-> Transmit PDO Mapping/SubIndex 014
//     PlcTask Inputs/P13_BottleTransfer.IaDataRobotREG[15] <-> Transmit PDO Mapping/SubIndex 015
//     PlcTask Inputs/P13_BottleTransfer.IaDataRobotREG[16] <-> Transmit PDO Mapping/SubIndex 016
//     PlcTask Inputs/P13_BottleTransfer.IaDataRobotREG[17] <-> Transmit PDO Mapping/SubIndex 017
//     PlcTask Inputs/P13_BottleTransfer.IaDataRobotREG[18] <-> Transmit PDO Mapping/SubIndex 018
//     PlcTask Inputs/P13_BottleTransfer.IaDataRobotREG[19] <-> Transmit PDO Mapping/SubIndex 019
//     PlcTask Inputs/P13_BottleTransfer.IaDataRobotREG[20] <-> Transmit PDO Mapping/SubIndex 020
//     PlcTask Inputs/P13_BottleTransfer.IaDataRobotREG[21] <-> Transmit PDO Mapping/SubIndex 021
//     PlcTask Inputs/P13_BottleTransfer.IaDataRobotREG[22] <-> Transmit PDO Mapping/SubIndex 022
//     PlcTask Inputs/P13_BottleTransfer.IaDataRobotREG[23] <-> Transmit PDO Mapping/SubIndex 023
//     PlcTask Inputs/P13_BottleTransfer.IaDataRobotREG[24] <-> Transmit PDO Mapping/SubIndex 024
//     PlcTask Inputs/P13_BottleTransfer.IaDataRobotREG[25] <-> Transmit PDO Mapping/SubIndex 025
//     PlcTask Inputs/P13_BottleTransfer.IaDataRobotREG[26] <-> Transmit PDO Mapping/SubIndex 026
//     PlcTask Inputs/P13_BottleTransfer.IaDataRobotREG[27] <-> Transmit PDO Mapping/SubIndex 027
//     PlcTask Inputs/P13_BottleTransfer.IaDataRobotREG[28] <-> Transmit PDO Mapping/SubIndex 028
//     PlcTask Inputs/P13_BottleTransfer.IaDataRobotREG[29] <-> Transmit PDO Mapping/SubIndex 029
//     PlcTask Inputs/P13_BottleTransfer.IaDataRobotREG[30] <-> Transmit PDO Mapping/SubIndex 030
//     PlcTask Inputs/P13_BottleTransfer.IaDataRobotREG[31] <-> Transmit PDO Mapping/SubIndex 031
//     PlcTask Inputs/P13_BottleTransfer.IaDataRobotREG[32] <-> Transmit PDO Mapping/SubIndex 032
//     PlcTask Inputs/P13_BottleTransfer.IaDataRobotREG[9] <-> Transmit PDO Mapping/SubIndex 009
//     PlcTask Inputs/P13_BottleTransfer.IaDataRobotREG[1] <-> Transmit PDO Mapping/SubIndex 001_1
//     PlcTask Inputs/P13_BottleTransfer.IaDataRobotREG[2] <-> Transmit PDO Mapping/SubIndex 002_1
//     PlcTask Inputs/P13_BottleTransfer.IaDataRobotREG[3] <-> Transmit PDO Mapping/SubIndex 003_1
//     PlcTask Inputs/P13_BottleTransfer.IaDataRobotREG[4] <-> Transmit PDO Mapping/SubIndex 004_1
//     PlcTask Inputs/P13_BottleTransfer.IaDataRobotREG[5] <-> Transmit PDO Mapping/SubIndex 005_1
//     PlcTask Inputs/P13_BottleTransfer.IaDataRobotREG[6] <-> Transmit PDO Mapping/SubIndex 006_1
//     PlcTask Inputs/P13_BottleTransfer.IaDataRobotREG[7] <-> Transmit PDO Mapping/SubIndex 007_1
//     PlcTask Inputs/P13_BottleTransfer.IaDataRobotREG[8] <-> Transmit PDO Mapping/SubIndex 008_1
//     PlcTask Outputs/P13_BottleTransfer.QaDataRobotIO[1] <-> Receive PDO Mapping/SubIndex 001
//     PlcTask Outputs/P13_BottleTransfer.QaDataRobotIO[2] <-> Receive PDO Mapping/SubIndex 002
//     PlcTask Outputs/P13_BottleTransfer.QaDataRobotIO[3] <-> Receive PDO Mapping/SubIndex 003
//     PlcTask Outputs/P13_BottleTransfer.QaDataRobotIO[4] <-> Receive PDO Mapping/SubIndex 004
//     PlcTask Outputs/P13_BottleTransfer.QaDataRobotIO[5] <-> Receive PDO Mapping/SubIndex 005
//     PlcTask Outputs/P13_BottleTransfer.QaDataRobotIO[6] <-> Receive PDO Mapping/SubIndex 006
//     PlcTask Outputs/P13_BottleTransfer.QaDataRobotIO[7] <-> Receive PDO Mapping/SubIndex 007
//     PlcTask Outputs/P13_BottleTransfer.QaDataRobotIO[8] <-> Receive PDO Mapping/SubIndex 008
//     PlcTask Outputs/P13_BottleTransfer.QaDataRobotREG[10] <-> Receive PDO Mapping/SubIndex 010
//     PlcTask Outputs/P13_BottleTransfer.QaDataRobotREG[11] <-> Receive PDO Mapping/SubIndex 011
//     PlcTask Outputs/P13_BottleTransfer.QaDataRobotREG[12] <-> Receive PDO Mapping/SubIndex 012
//     PlcTask Outputs/P13_BottleTransfer.QaDataRobotREG[13] <-> Receive PDO Mapping/SubIndex 013
//     PlcTask Outputs/P13_BottleTransfer.QaDataRobotREG[14] <-> Receive PDO Mapping/SubIndex 014
//     PlcTask Outputs/P13_BottleTransfer.QaDataRobotREG[15] <-> Receive PDO Mapping/SubIndex 015
//     PlcTask Outputs/P13_BottleTransfer.QaDataRobotREG[16] <-> Receive PDO Mapping/SubIndex 016
//     PlcTask Outputs/P13_BottleTransfer.QaDataRobotREG[17] <-> Receive PDO Mapping/SubIndex 017
//     PlcTask Outputs/P13_BottleTransfer.QaDataRobotREG[18] <-> Receive PDO Mapping/SubIndex 018
//     PlcTask Outputs/P13_BottleTransfer.QaDataRobotREG[19] <-> Receive PDO Mapping/SubIndex 019
//     PlcTask Outputs/P13_BottleTransfer.QaDataRobotREG[20] <-> Receive PDO Mapping/SubIndex 020
//     PlcTask Outputs/P13_BottleTransfer.QaDataRobotREG[21] <-> Receive PDO Mapping/SubIndex 021
//     PlcTask Outputs/P13_BottleTransfer.QaDataRobotREG[22] <-> Receive PDO Mapping/SubIndex 022
//     PlcTask Outputs/P13_BottleTransfer.QaDataRobotREG[23] <-> Receive PDO Mapping/SubIndex 023
//     PlcTask Outputs/P13_BottleTransfer.QaDataRobotREG[24] <-> Receive PDO Mapping/SubIndex 024
//     PlcTask Outputs/P13_BottleTransfer.QaDataRobotREG[25] <-> Receive PDO Mapping/SubIndex 025
//     PlcTask Outputs/P13_BottleTransfer.QaDataRobotREG[26] <-> Receive PDO Mapping/SubIndex 026
//     PlcTask Outputs/P13_BottleTransfer.QaDataRobotREG[27] <-> Receive PDO Mapping/SubIndex 027
//     PlcTask Outputs/P13_BottleTransfer.QaDataRobotREG[28] <-> Receive PDO Mapping/SubIndex 028
//     PlcTask Outputs/P13_BottleTransfer.QaDataRobotREG[29] <-> Receive PDO Mapping/SubIndex 029
//     PlcTask Outputs/P13_BottleTransfer.QaDataRobotREG[30] <-> Receive PDO Mapping/SubIndex 030
//     PlcTask Outputs/P13_BottleTransfer.QaDataRobotREG[31] <-> Receive PDO Mapping/SubIndex 031
//     PlcTask Outputs/P13_BottleTransfer.QaDataRobotREG[32] <-> Receive PDO Mapping/SubIndex 032
//     PlcTask Outputs/P13_BottleTransfer.QaDataRobotREG[9] <-> Receive PDO Mapping/SubIndex 009
//     PlcTask Outputs/P13_BottleTransfer.QaDataRobotREG[1] <-> Receive PDO Mapping/SubIndex 001_1
//     PlcTask Outputs/P13_BottleTransfer.QaDataRobotREG[2] <-> Receive PDO Mapping/SubIndex 002_1
//     PlcTask Outputs/P13_BottleTransfer.QaDataRobotREG[3] <-> Receive PDO Mapping/SubIndex 003_1
//     PlcTask Outputs/P13_BottleTransfer.QaDataRobotREG[4] <-> Receive PDO Mapping/SubIndex 004_1
//     PlcTask Outputs/P13_BottleTransfer.QaDataRobotREG[5] <-> Receive PDO Mapping/SubIndex 005_1
//     PlcTask Outputs/P13_BottleTransfer.QaDataRobotREG[6] <-> Receive PDO Mapping/SubIndex 006_1
//     PlcTask Outputs/P13_BottleTransfer.QaDataRobotREG[7] <-> Receive PDO Mapping/SubIndex 007_1
//     PlcTask Outputs/P13_BottleTransfer.QaDataRobotREG[8] <-> Receive PDO Mapping/SubIndex 008_1
//   (this object) <-> Device 1 (EtherCAT)/R2_242A1 (CU1128)/R2_242A1 (CU1128-B)/770A1 (EP6228-0022)
//     PlcTask Inputs/P00_ReadRFIDCard.AusiAfterDispencers2PhaseReaderInputData <-> Module 5 (IO-Link Slave)/IO-Link Port3_in/P00_ReadRFIDCard.AusiAfterDispencers2PhaseReaderInputData
//     PlcTask Inputs/P00_ReadRFIDCard.AusiAfterDispencersReaderInputData <-> Module 4 (IO-Link Slave)/IO-Link Port2_in/P00_ReadRFIDCard.AusiAfterDispencersReaderInputData
//     PlcTask Inputs/P00_ReadRFIDCard.AusiAfterScrewerReaderInputData <-> Module 9 (IO-Link Slave)/IO-Link Port7_in/P00_ReadRFIDCard.AusiAfterScrewerReaderInputData
//     PlcTask Inputs/P00_ReadRFIDCard.AusiBeforeScrewerReaderInputData <-> Module 8 (IO-Link Slave)/IO-Link Port6_in/P00_ReadRFIDCard.AusiBeforeScrewerReaderInputData
//     PlcTask Inputs/P00_ReadRFIDCard.AusiBottleTransferReaderInputData <-> Module 10 (IO-Link Slave)/IO-Link Port8_in/P00_ReadRFIDCard.AusiBottleTransferReaderInputData
//     PlcTask Inputs/P00_ReadRFIDCard.AusiCapSorterReaderInputData <-> Module 6 (IO-Link Slave)/IO-Link Port4_in/P00_ReadRFIDCard.AusiLidFeederReaderInputData
//     PlcTask Inputs/P00_ReadRFIDCard.AusiDispencerReaderInputData <-> Module 3 (IO-Link Slave)/IO-Link Port1_in/P00_ReadRFIDCard.AusiDispencerReaderInputData
//     PlcTask Inputs/P00_ReadRFIDCard.AusiLidSealerReaderInputData <-> Module 7 (IO-Link Slave)/IO-Link Port5_in/P00_ReadRFIDCard.AusiLidSealerReaderInputData
//     PlcTask Inputs/P00_ReadRFIDCard.IBAfterDispencers2PhaseReaderDataCounterIn <-> Module 5 (IO-Link Slave)/IO-Link Port3_in/P00_ReadRFIDCard.IBAfterDispencers2PhaseReaderDataCounterIn
//     PlcTask Inputs/P00_ReadRFIDCard.IBAfterDispencers2PhaseReaderErrorValue <-> Module 5 (IO-Link Slave)/IO-Link Port3_in/P00_ReadRFIDCard.IBAfterDispencers2PhaseReaderErrorValue
//     PlcTask Inputs/P00_ReadRFIDCard.IBAfterDispencersReaderDataCounterIn <-> Module 4 (IO-Link Slave)/IO-Link Port2_in/P00_ReadRFIDCard.IBAfterDispencersReaderDataCounterIn
//     PlcTask Inputs/P00_ReadRFIDCard.IBAfterDispencersReaderErrorValue <-> Module 4 (IO-Link Slave)/IO-Link Port2_in/P00_ReadRFIDCard.IBAfterDispencersReaderErrorValue
//     PlcTask Inputs/P00_ReadRFIDCard.IBAfterScrewerReaderDataCounterIn <-> Module 9 (IO-Link Slave)/IO-Link Port7_in/P00_ReadRFIDCard.IBAfterScrewerReaderDataCounterIn
//     PlcTask Inputs/P00_ReadRFIDCard.IBAfterScrewerReaderErrorValue <-> Module 9 (IO-Link Slave)/IO-Link Port7_in/P00_ReadRFIDCard.IBAfterScrewerReaderErrorValue
//     PlcTask Inputs/P00_ReadRFIDCard.IBBeforeScrewerReaderDataCounterIn <-> Module 8 (IO-Link Slave)/IO-Link Port6_in/P00_ReadRFIDCard.IBBeforeScrewerReaderDataCounterIn
//     PlcTask Inputs/P00_ReadRFIDCard.IBBeforeScrewerReaderErrorValue <-> Module 8 (IO-Link Slave)/IO-Link Port6_in/P00_ReadRFIDCard.IBBeforeScrewerReaderErrorValue
//     PlcTask Inputs/P00_ReadRFIDCard.IBBottleTransferReaderDataCounterIn <-> Module 10 (IO-Link Slave)/IO-Link Port8_in/P00_ReadRFIDCard.IBBottleTransferReaderDataCounterIn
//     PlcTask Inputs/P00_ReadRFIDCard.IBBottleTransferReaderErrorValue <-> Module 10 (IO-Link Slave)/IO-Link Port8_in/P00_ReadRFIDCard.IBBottleTransferReaderErrorValue
//     PlcTask Inputs/P00_ReadRFIDCard.IBCapSorterReaderDataCounterIn <-> Module 6 (IO-Link Slave)/IO-Link Port4_in/P00_ReadRFIDCard.IBLidFeederReaderDataCounterIn
//     PlcTask Inputs/P00_ReadRFIDCard.IBCapSorterReaderErrorValue <-> Module 6 (IO-Link Slave)/IO-Link Port4_in/P00_ReadRFIDCard.IBLidFeederReaderErrorValue
//     PlcTask Inputs/P00_ReadRFIDCard.IBDispencerReaderDataCounterIn <-> Module 3 (IO-Link Slave)/IO-Link Port1_in/P00_ReadRFIDCard.IBDispencerReaderDataCounterIn
//     PlcTask Inputs/P00_ReadRFIDCard.IBDispencerReaderErrorValue <-> Module 3 (IO-Link Slave)/IO-Link Port1_in/P00_ReadRFIDCard.IBDispencerReaderErrorValue
//     PlcTask Inputs/P00_ReadRFIDCard.IBLidSealerReaderDataCounterIn <-> Module 7 (IO-Link Slave)/IO-Link Port5_in/P00_ReadRFIDCard.IBLidSealerReaderDataCounterIn
//     PlcTask Inputs/P00_ReadRFIDCard.IBLidSealerReaderErrorValue <-> Module 7 (IO-Link Slave)/IO-Link Port5_in/P00_ReadRFIDCard.IBLidSealerReaderErrorValue
//     PlcTask Inputs/P00_ReadRFIDCard.IbAfterDispencers2PhaseReaderCmdEnd <-> Module 5 (IO-Link Slave)/IO-Link Port3_in/P00_ReadRFIDCard.IbAfterDispencers2PhaseReaderCmdEnd
//     PlcTask Inputs/P00_ReadRFIDCard.IbAfterDispencers2PhaseReaderCmdStartAck <-> Module 5 (IO-Link Slave)/IO-Link Port3_in/P00_ReadRFIDCard.IbAfterDispencers2PhaseReaderCmdStartAck
//     PlcTask Inputs/P00_ReadRFIDCard.IbAfterDispencers2PhaseReaderTagPresent <-> Module 5 (IO-Link Slave)/IO-Link Port3_in/P00_ReadRFIDCard.IbAfterDispencers2PhaseReaderTagPresent
//     PlcTask Inputs/P00_ReadRFIDCard.IbAfterDispencersReaderCmdEnd <-> Module 4 (IO-Link Slave)/IO-Link Port2_in/P00_ReadRFIDCard.IbAfterDispencersReaderCmdEnd
//     PlcTask Inputs/P00_ReadRFIDCard.IbAfterDispencersReaderCmdStartAck <-> Module 4 (IO-Link Slave)/IO-Link Port2_in/P00_ReadRFIDCard.IbAfterDispencersReaderCmdStartAck
//     PlcTask Inputs/P00_ReadRFIDCard.IbAfterDispencersReaderTagPresent <-> Module 4 (IO-Link Slave)/IO-Link Port2_in/P00_ReadRFIDCard.IbAfterDispencersReaderTagPresent
//     PlcTask Inputs/P00_ReadRFIDCard.IbAfterScrewerReaderCmdEnd <-> Module 9 (IO-Link Slave)/IO-Link Port7_in/P00_ReadRFIDCard.IbAfterScrewerReaderCmdEnd
//     PlcTask Inputs/P00_ReadRFIDCard.IbAfterScrewerReaderCmdStartAck <-> Module 9 (IO-Link Slave)/IO-Link Port7_in/P00_ReadRFIDCard.IbAfterScrewerReaderCmdStartAck
//     PlcTask Inputs/P00_ReadRFIDCard.IbAfterScrewerReaderTagPresent <-> Module 9 (IO-Link Slave)/IO-Link Port7_in/P00_ReadRFIDCard.IbAfterScrewerReaderTagPresent
//     PlcTask Inputs/P00_ReadRFIDCard.IbBeforeScrewerReaderCmdEnd <-> Module 8 (IO-Link Slave)/IO-Link Port6_in/P00_ReadRFIDCard.IbBeforeScrewerReaderCmdEnd
//     PlcTask Inputs/P00_ReadRFIDCard.IbBeforeScrewerReaderCmdStartAck <-> Module 8 (IO-Link Slave)/IO-Link Port6_in/P00_ReadRFIDCard.IbBeforeScrewerReaderCmdStartAck
//     PlcTask Inputs/P00_ReadRFIDCard.IbBeforeScrewerReaderTagPresent <-> Module 8 (IO-Link Slave)/IO-Link Port6_in/P00_ReadRFIDCard.IbBeforeScrewerReaderTagPresent
//     PlcTask Inputs/P00_ReadRFIDCard.IbBottleTransferReaderCmdEnd <-> Module 10 (IO-Link Slave)/IO-Link Port8_in/P00_ReadRFIDCard.IbBottleTransferReaderCmdEnd
//     PlcTask Inputs/P00_ReadRFIDCard.IbBottleTransferReaderCmdStartAck <-> Module 10 (IO-Link Slave)/IO-Link Port8_in/P00_ReadRFIDCard.IbBottleTransferReaderCmdStartAck
//     PlcTask Inputs/P00_ReadRFIDCard.IbBottleTransferReaderTagPresent <-> Module 10 (IO-Link Slave)/IO-Link Port8_in/P00_ReadRFIDCard.IbBottleTransferReaderTagPresent
//     PlcTask Inputs/P00_ReadRFIDCard.IbCapSorterReaderCmdEnd <-> Module 6 (IO-Link Slave)/IO-Link Port4_in/P00_ReadRFIDCard.IbLidFeederReaderCmdEnd
//     PlcTask Inputs/P00_ReadRFIDCard.IbCapSorterReaderCmdStartAck <-> Module 6 (IO-Link Slave)/IO-Link Port4_in/P00_ReadRFIDCard.IbLidFeederReaderCmdStartAck
//     PlcTask Inputs/P00_ReadRFIDCard.IbCapSorterReaderTagPresent <-> Module 6 (IO-Link Slave)/IO-Link Port4_in/P00_ReadRFIDCard.IbLidFeederReaderTagPresent
//     PlcTask Inputs/P00_ReadRFIDCard.IbDispencerReaderCmdEnd <-> Module 3 (IO-Link Slave)/IO-Link Port1_in/P00_ReadRFIDCard.IbDispencerReaderCmdEnd
//     PlcTask Inputs/P00_ReadRFIDCard.IbDispencerReaderCmdStartAck <-> Module 3 (IO-Link Slave)/IO-Link Port1_in/P00_ReadRFIDCard.IbDispencerReaderCmdStartAck
//     PlcTask Inputs/P00_ReadRFIDCard.IbDispencerReaderTagPresent <-> Module 3 (IO-Link Slave)/IO-Link Port1_in/P00_ReadRFIDCard.IbDispencerReaderTagPresent
//     PlcTask Inputs/P00_ReadRFIDCard.IbLidSealerReaderCmdEnd <-> Module 7 (IO-Link Slave)/IO-Link Port5_in/P00_ReadRFIDCard.IbLidSealerReaderCmdEnd
//     PlcTask Inputs/P00_ReadRFIDCard.IbLidSealerReaderCmdStartAck <-> Module 7 (IO-Link Slave)/IO-Link Port5_in/P00_ReadRFIDCard.IbLidSealerReaderCmdStartAck
//     PlcTask Inputs/P00_ReadRFIDCard.IbLidSealerReaderTagPresent <-> Module 7 (IO-Link Slave)/IO-Link Port5_in/P00_ReadRFIDCard.IbLidSealerReaderTagPresent
//     PlcTask Outputs/P00_ReadRFIDCard.AusiAfterDispencers2PhaseReaderOutputData <-> Module 5 (IO-Link Slave)/IO-Link Port3_out/P00_ReadRFIDCard.AusiAfterDispencers2PhaseReaderOutputData
//     PlcTask Outputs/P00_ReadRFIDCard.AusiAfterDispencersReaderOutputData <-> Module 4 (IO-Link Slave)/IO-Link Port2_out/P00_ReadRFIDCard.AusiAfterDispencersReaderOutputData
//     PlcTask Outputs/P00_ReadRFIDCard.AusiAfterScrewerReaderOutputData <-> Module 9 (IO-Link Slave)/IO-Link Port7_out/P00_ReadRFIDCard.AusiAfterScrewerReaderOutputData
//     PlcTask Outputs/P00_ReadRFIDCard.AusiBeforeScrewerReaderOutputData <-> Module 8 (IO-Link Slave)/IO-Link Port6_out/P00_ReadRFIDCard.AusiBeforeScrewerReaderOutputData
//     PlcTask Outputs/P00_ReadRFIDCard.AusiBottleTransferReaderOutputData <-> Module 10 (IO-Link Slave)/IO-Link Port8_out/P00_ReadRFIDCard.AusiBottleTransferReaderOutputData
//     PlcTask Outputs/P00_ReadRFIDCard.AusiCapSorterReaderOutputData <-> Module 6 (IO-Link Slave)/IO-Link Port4_out/P00_ReadRFIDCard.AusiLidFeederReaderOutputData
//     PlcTask Outputs/P00_ReadRFIDCard.AusiDispencerReaderOutputData <-> Module 3 (IO-Link Slave)/IO-Link Port1_out/P00_ReadRFIDCard.AusiDispencerReaderOutputData
//     PlcTask Outputs/P00_ReadRFIDCard.AusiLidSealerReaderOutputData <-> Module 7 (IO-Link Slave)/IO-Link Port5_out/P00_ReadRFIDCard.AusiLidSealerReaderOutputData
//     PlcTask Outputs/P00_ReadRFIDCard.IBAfterDispencers2PhaseReaderCmmandValue <-> Module 5 (IO-Link Slave)/IO-Link Port3_out/P00_ReadRFIDCard.IBAfterDispencers2PhaseReaderCmmandValue
//     PlcTask Outputs/P00_ReadRFIDCard.IBAfterDispencers2PhaseReaderDataCounterOut <-> Module 5 (IO-Link Slave)/IO-Link Port3_out/P00_ReadRFIDCard.IBAfterDispencers2PhaseReaderDataCounterOut
//     PlcTask Outputs/P00_ReadRFIDCard.IBAfterDispencersReaderCmmandValue <-> Module 4 (IO-Link Slave)/IO-Link Port2_out/P00_ReadRFIDCard.IBAfterDispencersReaderCmmandValue
//     PlcTask Outputs/P00_ReadRFIDCard.IBAfterDispencersReaderDataCounterOut <-> Module 4 (IO-Link Slave)/IO-Link Port2_out/P00_ReadRFIDCard.IBAfterDispencersReaderDataCounterOut
//     PlcTask Outputs/P00_ReadRFIDCard.IBAfterScrewerReaderCmmandValue <-> Module 9 (IO-Link Slave)/IO-Link Port7_out/P00_ReadRFIDCard.IBAfterScrewerReaderCmmandValue
//     PlcTask Outputs/P00_ReadRFIDCard.IBAfterScrewerReaderDataCounterOut <-> Module 9 (IO-Link Slave)/IO-Link Port7_out/P00_ReadRFIDCard.IBAfterScrewerReaderDataCounterOut
//     PlcTask Outputs/P00_ReadRFIDCard.IBBeforeScrewerReaderCmmandValue <-> Module 8 (IO-Link Slave)/IO-Link Port6_out/P00_ReadRFIDCard.IBBeforeScrewerReaderCmmandValue
//     PlcTask Outputs/P00_ReadRFIDCard.IBBeforeScrewerReaderDataCounterOut <-> Module 8 (IO-Link Slave)/IO-Link Port6_out/P00_ReadRFIDCard.IBBeforeScrewerReaderDataCounterOut
//     PlcTask Outputs/P00_ReadRFIDCard.IBBottleTransferReaderCmmandValue <-> Module 10 (IO-Link Slave)/IO-Link Port8_out/P00_ReadRFIDCard.IBBottleTransferReaderCmmandValue
//     PlcTask Outputs/P00_ReadRFIDCard.IBBottleTransferReaderDataCounterOut <-> Module 10 (IO-Link Slave)/IO-Link Port8_out/P00_ReadRFIDCard.IBBottleTransferReaderDataCounterOut
//     PlcTask Outputs/P00_ReadRFIDCard.IBCapSorterReaderCmmandValue <-> Module 6 (IO-Link Slave)/IO-Link Port4_out/P00_ReadRFIDCard.IBLidFeederReaderCmmandValue
//     PlcTask Outputs/P00_ReadRFIDCard.IBCapSorterReaderDataCounterOut <-> Module 6 (IO-Link Slave)/IO-Link Port4_out/P00_ReadRFIDCard.IBLidFeederReaderDataCounterOut
//     PlcTask Outputs/P00_ReadRFIDCard.IBDispencerReaderCmmandValue <-> Module 3 (IO-Link Slave)/IO-Link Port1_out/P00_ReadRFIDCard.IBDispencerReaderCmmandValue
//     PlcTask Outputs/P00_ReadRFIDCard.IBDispencerReaderDataCounterOut <-> Module 3 (IO-Link Slave)/IO-Link Port1_out/P00_ReadRFIDCard.IBDispencerReaderDataCounterOut
//     PlcTask Outputs/P00_ReadRFIDCard.IBLidSealerReaderCmmandValue <-> Module 7 (IO-Link Slave)/IO-Link Port5_out/P00_ReadRFIDCard.IBLidSealerReaderCmmandValue
//     PlcTask Outputs/P00_ReadRFIDCard.IBLidSealerReaderDataCounterOut <-> Module 7 (IO-Link Slave)/IO-Link Port5_out/P00_ReadRFIDCard.IBLidSealerReaderDataCounterOut
//     PlcTask Outputs/P00_ReadRFIDCard.IbAfterDispencers2PhaseReaderCmdStart <-> Module 5 (IO-Link Slave)/IO-Link Port3_out/P00_ReadRFIDCard.IbAfterDispencers2PhaseReaderCmdStart
//     PlcTask Outputs/P00_ReadRFIDCard.IbAfterDispencersReaderCmdStart <-> Module 4 (IO-Link Slave)/IO-Link Port2_out/P00_ReadRFIDCard.IbAfterDispencersReaderCmdStart
//     PlcTask Outputs/P00_ReadRFIDCard.IbAfterScrewerReaderCmdStart <-> Module 9 (IO-Link Slave)/IO-Link Port7_out/P00_ReadRFIDCard.IbAfterScrewerReaderCmdStart
//     PlcTask Outputs/P00_ReadRFIDCard.IbBeforeScrewerReaderCmdStart <-> Module 8 (IO-Link Slave)/IO-Link Port6_out/P00_ReadRFIDCard.IbBeforeScrewerReaderCmdStart
//     PlcTask Outputs/P00_ReadRFIDCard.IbBottleTransferReaderCmdStart <-> Module 10 (IO-Link Slave)/IO-Link Port8_out/P00_ReadRFIDCard.IbBottleTransferReaderCmdStart
//     PlcTask Outputs/P00_ReadRFIDCard.IbCapSorterReaderCmdStart <-> Module 6 (IO-Link Slave)/IO-Link Port4_out/P00_ReadRFIDCard.IbLidFeederReaderCmdStart
//     PlcTask Outputs/P00_ReadRFIDCard.IbDispencerReaderCmdStart <-> Module 3 (IO-Link Slave)/IO-Link Port1_out/P00_ReadRFIDCard.IbDispencerReaderCmdStart
//     PlcTask Outputs/P00_ReadRFIDCard.IbLidSealerReaderCmdStart <-> Module 7 (IO-Link Slave)/IO-Link Port5_out/P00_ReadRFIDCard.IbLidSealerReaderCmdStart
//   (this object) <-> Device 1 (EtherCAT)/R2_242A1 (CU1128)/R2_242A1 (CU1128-B)/Box 27 (EP6228-0022)
//     PlcTask Inputs/P00_ReadRFIDCard.AusiLidFeederReaderInputData <-> Module 4 (IO-Link Slave)/IO-Link Port2_in/Input data
//     PlcTask Inputs/P00_ReadRFIDCard.IBLidFeederReaderDataCounterIn <-> Module 4 (IO-Link Slave)/IO-Link Port2_in/Data / Block counter
//     PlcTask Inputs/P00_ReadRFIDCard.IBLidFeederReaderErrorValue <-> Module 4 (IO-Link Slave)/IO-Link Port2_in/Error value
//     PlcTask Inputs/P00_ReadRFIDCard.IbLidFeederReaderCmdEnd <-> Module 4 (IO-Link Slave)/IO-Link Port2_in/Cmd End
//     PlcTask Inputs/P00_ReadRFIDCard.IbLidFeederReaderCmdStartAck <-> Module 4 (IO-Link Slave)/IO-Link Port2_in/Cmd Start Acknowledge
//     PlcTask Inputs/P00_ReadRFIDCard.IbLidFeederReaderTagPresent <-> Module 4 (IO-Link Slave)/IO-Link Port2_in/Tag Present
//     PlcTask Inputs/P09_CapPuttedCheck.IbCapPuttedCheckSensorError_Wenglor <-> Module 3 (IO-Link Slave)/IO-Link Port1_in/Error
//     PlcTask Inputs/P09_CapPuttedCheck.IbCapPuttedCheckSensorSSC1_Wenglor <-> Module 3 (IO-Link Slave)/IO-Link Port1_in/SSC1 - Switching Signal 1
//     PlcTask Inputs/P09_CapPuttedCheck.IbCapPuttedCheckSensorSSC2_Wenglor <-> Module 3 (IO-Link Slave)/IO-Link Port1_in/SSC2 - Switching Signal 2
//     PlcTask Inputs/P09_CapPuttedCheck.IbCapPuttedCheckSensorScale_Wenglor <-> Module 3 (IO-Link Slave)/IO-Link Port1_in/Scale
//     PlcTask Inputs/P09_CapPuttedCheck.IbCapPuttedCheckSensorWarning_1_Wenglor <-> Module 3 (IO-Link Slave)/IO-Link Port1_in/Indication Warning/Error 1
//     PlcTask Inputs/P09_CapPuttedCheck.IbCapPuttedCheckSensorWarning_2_Wenglor <-> Module 3 (IO-Link Slave)/IO-Link Port1_in/Indication Warning/Error 2
//     PlcTask Inputs/P09_CapPuttedCheck.IbCapPuttedCheckSensorWarning_3_Wenglor <-> Module 3 (IO-Link Slave)/IO-Link Port1_in/Indication Warning/Error 3
//     PlcTask Inputs/P09_CapPuttedCheck.IbCapPuttedCheckSensorWarning_4_Wenglor <-> Module 3 (IO-Link Slave)/IO-Link Port1_in/Indication Warning/Error 4
//     PlcTask Inputs/P09_CapPuttedCheck.IbCapPuttedCheckSensorWarning_Wenglor <-> Module 3 (IO-Link Slave)/IO-Link Port1_in/Warning
//     PlcTask Inputs/P09_CapPuttedCheck.IdiCapPuttedCheckSensorCV_Wenglor <-> Module 3 (IO-Link Slave)/IO-Link Port1_in/Measurement value: Distance
//     PlcTask Inputs/P11_RollerScrewer.AusiReaderInputData <-> Module 5 (IO-Link Slave)/IO-Link Port3_in/Input data
//     PlcTask Inputs/P11_RollerScrewer.IBReaderDataCounterIn <-> Module 5 (IO-Link Slave)/IO-Link Port3_in/Data / Block counter
//     PlcTask Inputs/P11_RollerScrewer.IBReaderErrorValue <-> Module 5 (IO-Link Slave)/IO-Link Port3_in/Error value
//     PlcTask Inputs/P11_RollerScrewer.IbReaderCmdEnd <-> Module 5 (IO-Link Slave)/IO-Link Port3_in/Cmd End
//     PlcTask Inputs/P11_RollerScrewer.IbReaderCmdStartAck <-> Module 5 (IO-Link Slave)/IO-Link Port3_in/Cmd Start Acknowledge
//     PlcTask Inputs/P11_RollerScrewer.IbReaderTagPresent <-> Module 5 (IO-Link Slave)/IO-Link Port3_in/Tag Present
//     PlcTask Outputs/P00_ReadRFIDCard.AusiLidFeederReaderOutputData <-> Module 4 (IO-Link Slave)/IO-Link Port2_out/Output data
//     PlcTask Outputs/P00_ReadRFIDCard.IBLidFeederReaderCmmandValue <-> Module 4 (IO-Link Slave)/IO-Link Port2_out/Command value
//     PlcTask Outputs/P00_ReadRFIDCard.IBLidFeederReaderDataCounterOut <-> Module 4 (IO-Link Slave)/IO-Link Port2_out/Data / Block counter
//     PlcTask Outputs/P00_ReadRFIDCard.IbLidFeederReaderCmdStart <-> Module 4 (IO-Link Slave)/IO-Link Port2_out/Cmd Start
//     PlcTask Outputs/P09_CapPuttedCheck.QbCapPuttedCheckSensorControlSignal_Wenglor <-> Module 3 (IO-Link Slave)/IO-Link Port1_out/Emitted Light
//     PlcTask Outputs/P09_CapPuttedCheck.QbCapPuttedCheckSensorFindMe_Wenglor <-> Module 3 (IO-Link Slave)/IO-Link Port1_out/Find Me
//     PlcTask Outputs/P09_CapPuttedCheck.QbCapPuttedCheckSensorTeachSSC1_Wenglor <-> Module 3 (IO-Link Slave)/IO-Link Port1_out/SSC1 Teach-In
//     PlcTask Outputs/P09_CapPuttedCheck.QbCapPuttedCheckSensorTeachSSC2_Wenglor <-> Module 3 (IO-Link Slave)/IO-Link Port1_out/SSC2 Teach-In
//     PlcTask Outputs/P11_RollerScrewer.AusiReaderOutputData <-> Module 5 (IO-Link Slave)/IO-Link Port3_out/Output data
//     PlcTask Outputs/P11_RollerScrewer.IBReaderCmmandValue <-> Module 5 (IO-Link Slave)/IO-Link Port3_out/Command value
//     PlcTask Outputs/P11_RollerScrewer.IBReaderDataCounterOut <-> Module 5 (IO-Link Slave)/IO-Link Port3_out/Data / Block counter
//     PlcTask Outputs/P11_RollerScrewer.IbReaderCmdStart <-> Module 5 (IO-Link Slave)/IO-Link Port3_out/Cmd Start
//   (this object) <-> Device 1 (EtherCAT)/R2_242A1 (CU1128)/R2_242A1 (CU1128-B)/R2_641N1 (EtherCAT EB80 series)
//     PlcTask Inputs/P00_PneumaticValves.IABPneumatic641PressureRegulator[1] <-> 1. TxPDO/P00_PneumaticValves.IABPneumatic641PressureRegulator[1]
//     PlcTask Inputs/P00_PneumaticValves.IABPneumatic641PressureRegulator[2] <-> 1. TxPDO/P00_PneumaticValves.IABPneumatic641PressureRegulator[2]
//     PlcTask Inputs/P00_PneumaticValves.IABPneumatic641_N11AnalogInput1[1] <-> 1. TxPDO/Analogue Input Channel 1 (Byte1)
//     PlcTask Inputs/P00_PneumaticValves.IABPneumatic641_N11AnalogInput1[2] <-> 1. TxPDO/Analogue Input Channel 1 (Byte2)
//     PlcTask Inputs/P00_PneumaticValves.IABPneumatic641_N11AnalogInput2[1] <-> 1. TxPDO/Analogue Input Channel 2 (Byte1)
//     PlcTask Inputs/P00_PneumaticValves.IABPneumatic641_N11AnalogInput2[2] <-> 1. TxPDO/Analogue Input Channel 2 (Byte2)
//     PlcTask Inputs/P00_PneumaticValves.IABPneumatic641_N11AnalogInput3[1] <-> 1. TxPDO/Analogue Input Channel 3 (Byte1)
//     PlcTask Inputs/P00_PneumaticValves.IABPneumatic641_N11AnalogInput3[2] <-> 1. TxPDO/Analogue Input Channel 3 (Byte2)
//     PlcTask Inputs/P00_PneumaticValves.IABPneumatic641_N11AnalogInput4[1] <-> 1. TxPDO/Analogue Input Channel 4 (Byte1)
//     PlcTask Inputs/P00_PneumaticValves.IABPneumatic641_N11AnalogInput4[2] <-> 1. TxPDO/Analogue Input Channel 4 (Byte2)
//     PlcTask Inputs/P00_PneumaticValves.IABPneumatic641_N12DigitalInput <-> 1. TxPDO/8 Digital Input 1-8
//     PlcTask Outputs/P00_PneumaticValves.QABPneumatic641PressureRegulator[1] <-> 1. RxPDO/P00_PneumaticValves.QABPneumatic641PressureRegulator[1]
//     PlcTask Outputs/P00_PneumaticValves.QABPneumatic641PressureRegulator[2] <-> 1. RxPDO/P00_PneumaticValves.QABPneumatic641PressureRegulator[2]
//     PlcTask Outputs/P00_PneumaticValves.QABPneumatic641ValveCoils[1] <-> 1. RxPDO/P00_PneumaticValves.QABPneumatic641ValveCoils[1]
//     PlcTask Outputs/P00_PneumaticValves.QABPneumatic641ValveCoils[2] <-> 1. RxPDO/P00_PneumaticValves.QABPneumatic641ValveCoils[2]
//     PlcTask Outputs/P00_PneumaticValves.QABPneumatic641ValveCoils[3] <-> 1. RxPDO/P00_PneumaticValves.QABPneumatic641ValveCoils[3]
//     PlcTask Outputs/P00_PneumaticValves.QABPneumatic641ValveCoils[4] <-> 1. RxPDO/P00_PneumaticValves.QABPneumatic641ValveCoils[4]
//     PlcTask Outputs/P00_PneumaticValves.QABPneumatic641ValveCoils[5] <-> 1. RxPDO/P00_PneumaticValves.QABPneumatic641ValveCoils[5]
//     PlcTask Outputs/P00_PneumaticValves.QABPneumatic641ValveCoils[6] <-> 1. RxPDO/P00_PneumaticValves.QABPneumatic641ValveCoils[6]
//   (this object) <-> Device 1 (EtherCAT)/R2_242A1 (CU1128)/R2_242A1 (CU1128-B)/R2_642N1 (EtherCAT EB80 series)
//     PlcTask Inputs/P00_PneumaticValves.IABPneumatic642_N11DigitalInput <-> 1. TxPDO/P00_PneumaticValves.IABPneumatic642_N11DigitalInput
//     PlcTask Inputs/P00_PneumaticValves.IABPneumatic642_N13DigitalInput <-> 1. TxPDO/P00_PneumaticValves.IABPneumatic642_N13DigitalInput
//     PlcTask Inputs/P00_PneumaticValves.IABPneumatic642_N12DigitalInput <-> 1. TxPDO/P00_PneumaticValves.IABPneumatic642_N12DigitalInput
//     PlcTask Outputs/P00_PneumaticValves.QABPneumatic642ValveCoils[1] <-> 1. RxPDO/P00_PneumaticValves.QABPneumatic642ValveCoils[1]
//     PlcTask Outputs/P00_PneumaticValves.QABPneumatic642ValveCoils[2] <-> 1. RxPDO/P00_PneumaticValves.QABPneumatic642ValveCoils[2]
//     PlcTask Outputs/P00_PneumaticValves.QABPneumatic642ValveCoils[3] <-> 1. RxPDO/P00_PneumaticValves.QABPneumatic642ValveCoils[3]
//     PlcTask Outputs/P00_PneumaticValves.QABPneumatic642ValveCoils[4] <-> 1. RxPDO/P00_PneumaticValves.QABPneumatic642ValveCoils[4]
//     PlcTask Outputs/P00_PneumaticValves.QABPneumatic642ValveCoils[5] <-> 1. RxPDO/P00_PneumaticValves.QABPneumatic642ValveCoils[5]
//   (this object) <-> Device 1 (EtherCAT)/R2_242A1 (CU1128)/R2_242A1 (CU1128-B)/R2_643N1 (EtherCAT EB80 series)
//     PlcTask Inputs/P00_PneumaticValves.IABPneumatic643_N11DigitalInput <-> 1. TxPDO/P00_PneumaticValves.IABPneumatic643_N11DigitalInput
//     PlcTask Inputs/P00_PneumaticValves.IABPneumatic643_N12DigitalInput <-> 1. TxPDO/P00_PneumaticValves.IABPneumatic643_N12DigitalInput
//     PlcTask Inputs/P00_PneumaticValves.IABPneumatic643_N13DigitalInput <-> 1. TxPDO/P00_PneumaticValves.IABPneumatic643_N13DigitalInput
//     PlcTask Outputs/P00_PneumaticValves.QABPneumatic643ValveCoils[1] <-> 1. RxPDO/P00_PneumaticValves.QABPneumatic643ValveCoils[1]
//     PlcTask Outputs/P00_PneumaticValves.QABPneumatic643ValveCoils[2] <-> 1. RxPDO/P00_PneumaticValves.QABPneumatic643ValveCoils[2]
//     PlcTask Outputs/P00_PneumaticValves.QABPneumatic643ValveCoils[3] <-> 1. RxPDO/P00_PneumaticValves.QABPneumatic643ValveCoils[3]
//     PlcTask Outputs/P00_PneumaticValves.QABPneumatic643ValveCoils[4] <-> 1. RxPDO/P00_PneumaticValves.QABPneumatic643ValveCoils[4]
//     PlcTask Outputs/P00_PneumaticValves.QABPneumatic643ValveCoils[5] <-> 1. RxPDO/P00_PneumaticValves.QABPneumatic643ValveCoils[5]
//   (this object) <-> Device 1 (EtherCAT)/R2_242A1 (CU1128)/R2_242A1 (CU1128-B)/R2_644N1 (EtherCAT EB80 series)
//     PlcTask Inputs/P00_PneumaticValves.IABPneumatic644_N11DigitalInput <-> 1. TxPDO/P00_PneumaticValves.IABPneumatic644_N11DigitalInput
//     PlcTask Inputs/P00_PneumaticValves.IABPneumatic644_N12DigitalInput <-> 1. TxPDO/P00_PneumaticValves.IABPneumatic644_N12DigitalInput
//     PlcTask Inputs/P00_PneumaticValves.IABPneumatic644_N13DigitalInput <-> 1. TxPDO/P00_PneumaticValves.IABPneumatic644_N13DigitalInput
//     PlcTask Outputs/P00_PneumaticValves.QABPneumatic644ValveCoils[1] <-> 1. RxPDO/P00_PneumaticValves.QABPneumatic644ValveCoils[1]
//     PlcTask Outputs/P00_PneumaticValves.QABPneumatic644ValveCoils[2] <-> 1. RxPDO/P00_PneumaticValves.QABPneumatic644ValveCoils[2]
//     PlcTask Outputs/P00_PneumaticValves.QABPneumatic644ValveCoils[3] <-> 1. RxPDO/P00_PneumaticValves.QABPneumatic644ValveCoils[3]
//     PlcTask Outputs/P00_PneumaticValves.QABPneumatic644ValveCoils[4] <-> 1. RxPDO/P00_PneumaticValves.QABPneumatic644ValveCoils[4]
//     PlcTask Outputs/P00_PneumaticValves.QABPneumatic644ValveCoils[5] <-> 1. RxPDO/P00_PneumaticValves.QABPneumatic644ValveCoils[5]
//   (this object) <-> Device 1 (EtherCAT)/R2_242A1 (CU1128)/R2_242A1 (CU1128-B)/R2_645N1 (EtherCAT EB80 series)
//     PlcTask Inputs/P00_PneumaticValves.IABPneumatic645_1PressureRegulator[1] <-> 1. TxPDO/P00_PneumaticValves.IABPneumatic645_1PressureRegulator[1]
//     PlcTask Inputs/P00_PneumaticValves.IABPneumatic645_1PressureRegulator[2] <-> 1. TxPDO/P00_PneumaticValves.IABPneumatic645_1PressureRegulator[2]
//     PlcTask Inputs/P00_PneumaticValves.IABPneumatic645_2PressureRegulator[1] <-> 1. TxPDO/P00_PneumaticValves.IABPneumatic645_2PressureRegulator[1]
//     PlcTask Inputs/P00_PneumaticValves.IABPneumatic645_2PressureRegulator[2] <-> 1. TxPDO/P00_PneumaticValves.IABPneumatic645_2PressureRegulator[2]
//     PlcTask Inputs/P00_PneumaticValves.IABPneumatic645_N11AnalogInput1[1] <-> 1. TxPDO/P00_PneumaticValves.IABPneumatic645_N11AnalogInput1[1]
//     PlcTask Inputs/P00_PneumaticValves.IABPneumatic645_N11AnalogInput1[2] <-> 1. TxPDO/P00_PneumaticValves.IABPneumatic645_N11AnalogInput1[2]
//     PlcTask Inputs/P00_PneumaticValves.IABPneumatic645_N11AnalogInput2[1] <-> 1. TxPDO/P00_PneumaticValves.IABPneumatic645_N11AnalogInput2[1]
//     PlcTask Inputs/P00_PneumaticValves.IABPneumatic645_N11AnalogInput2[2] <-> 1. TxPDO/P00_PneumaticValves.IABPneumatic645_N11AnalogInput2[2]
//     PlcTask Inputs/P00_PneumaticValves.IABPneumatic645_N11AnalogInput3[1] <-> 1. TxPDO/P00_PneumaticValves.IABPneumatic645_N11AnalogInput3[1]
//     PlcTask Inputs/P00_PneumaticValves.IABPneumatic645_N11AnalogInput3[2] <-> 1. TxPDO/P00_PneumaticValves.IABPneumatic645_N11AnalogInput3[2]
//     PlcTask Inputs/P00_PneumaticValves.IABPneumatic645_N11AnalogInput4[1] <-> 1. TxPDO/P00_PneumaticValves.IABPneumatic645_N11AnalogInput4[1]
//     PlcTask Inputs/P00_PneumaticValves.IABPneumatic645_N11AnalogInput4[2] <-> 1. TxPDO/P00_PneumaticValves.IABPneumatic645_N11AnalogInput4[2]
//     PlcTask Inputs/P00_PneumaticValves.IABPneumatic645_N12DigitalInput <-> 1. TxPDO/8 Digital Input 1-8
//     PlcTask Outputs/P00_PneumaticValves.QABPneumatic645ValveCoils[1] <-> 1. RxPDO/Valve coils 1
//     PlcTask Outputs/P00_PneumaticValves.QABPneumatic645ValveCoils[2] <-> 1. RxPDO/Valve coils 2
//     PlcTask Outputs/P00_PneumaticValves.QABPneumatic645_1PressureRegulator[1] <-> 1. RxPDO/P00_PneumaticValves.QABPneumatic645_1PressureRegulator[1]
//     PlcTask Outputs/P00_PneumaticValves.QABPneumatic645_1PressureRegulator[2] <-> 1. RxPDO/P00_PneumaticValves.QABPneumatic645_1PressureRegulator[2]
//     PlcTask Outputs/P00_PneumaticValves.QABPneumatic645_2PressureRegulator[1] <-> 1. RxPDO/P00_PneumaticValves.QABPneumatic645_2PressureRegulator[1]
//     PlcTask Outputs/P00_PneumaticValves.QABPneumatic645_2PressureRegulator[2] <-> 1. RxPDO/P00_PneumaticValves.QABPneumatic645_2PressureRegulator[2]
//   (this object) <-> Device 1 (EtherCAT)/R2_242A1 (CU1128)/R2_242A1 (CU1128-B)/R2_647N1 (UCF) (EtherCat EB80 series)
//     PlcTask Inputs/P00_PneumaticValves.IABPneumatic647_N11DigitalInput <-> 1. TxPDO/P00_PneumaticValves.IABPneumatic647_N11DigitalInput
//     PlcTask Inputs/P00_PneumaticValves.IABPneumatic647_N12DigitalInput <-> 1. TxPDO/P00_PneumaticValves.IABPneumatic647_N12DigitalInput
//     PlcTask Outputs/P00_PneumaticValves.QABPneumatic647ValveCoils[1] <-> 1. RxPDO/P00_PneumaticValves.QABPneumatic644ValveCoils[1]
//     PlcTask Outputs/P00_PneumaticValves.QABPneumatic647ValveCoils[2] <-> 1. RxPDO/P00_PneumaticValves.QABPneumatic644ValveCoils[2]
//     PlcTask Outputs/P00_PneumaticValves.QABPneumatic647ValveCoils[3] <-> 1. RxPDO/P00_PneumaticValves.QABPneumatic644ValveCoils[3]
//     PlcTask Outputs/P00_PneumaticValves.QABPneumatic647ValveCoils[4] <-> 1. RxPDO/P00_PneumaticValves.QABPneumatic644ValveCoils[4]
//     PlcTask Outputs/P00_PneumaticValves.QABPneumatic647ValveCoils[5] <-> 1. RxPDO/P00_PneumaticValves.QABPneumatic644ValveCoils[5]
//   (this object) <-> Device 1 (EtherCAT)/R2_242A1 (CU1128)/R2_242A1 (CU1128-B)/R2_648N1 (za rob.) (EtherCat EB80 serier)
//     PlcTask Inputs/P13_BottleTransferAfterDrag.IABPneumatic648DigitalInput[1] <-> 1. TxPDO/P00_PneumaticValves.IABPneumatic644_N11DigitalInput
//     PlcTask Inputs/P13_BottleTransferAfterDrag.IABPneumatic648DigitalInput[2] <-> 1. TxPDO/P00_PneumaticValves.IABPneumatic644_N12DigitalInput
//     PlcTask Inputs/P13_BottleTransferAfterDrag.IABPneumatic648DigitalInput[3] <-> 1. TxPDO/P00_PneumaticValves.IABPneumatic644_N13DigitalInput
//     PlcTask Inputs/P13_BottleTransferAfterDrag.IABPneumatic648DigitalInput[4] <-> 1. TxPDO/8 Digital Input 25-32
//     PlcTask Outputs/P13_BottleTransferAfterDrag.QABPneumatic648ValveCoils[1] <-> 1. RxPDO/P00_PneumaticValves.QABPneumatic644ValveCoils[1]
//     PlcTask Outputs/P13_BottleTransferAfterDrag.QABPneumatic648ValveCoils[2] <-> 1. RxPDO/P00_PneumaticValves.QABPneumatic644ValveCoils[2]
//     PlcTask Outputs/P13_BottleTransferAfterDrag.QABPneumatic648ValveCoils[3] <-> 1. RxPDO/P00_PneumaticValves.QABPneumatic644ValveCoils[3]
//     PlcTask Outputs/P13_BottleTransferAfterDrag.QABPneumatic648ValveCoils[4] <-> 1. RxPDO/P00_PneumaticValves.QABPneumatic644ValveCoils[4]
//     PlcTask Outputs/P13_BottleTransferAfterDrag.QABPneumatic648ValveCoils[5] <-> 1. RxPDO/P00_PneumaticValves.QABPneumatic644ValveCoils[5]
//   (this object) <-> Device 1 (EtherCAT)/R2_242A1 (CU1128)/R2_242A1 (CU1128-B)/RC40_60A2 (EtherCAT EB80 series)
//     PlcTask Outputs/P11_RollerScrewer.QABPneumaticRollerScrewerValveCoils[{1..5}] <-> 1. RxPDO/Valve coils {1..33 step 8}-{8..40 step 8}  (5 links)
//   (this object) <-> Device 1 (EtherCAT)/R2_242A1 (CU1128)/R2_242A1 (CU1128-B)/RC40_BC1(EK1814)/RC40_DO1 (EL2008)
//     PlcTask Outputs/P00_Signalization.QbResetLamp <-> Channel 6/P00_Signalization.QbResetLamp
//   (this object) <-> Device 1 (EtherCAT)/R2_242A1 (CU1128)/R2_242A1 (CU1128-C)/PI_641N1 (EtherCAT EB80 series)
//     PlcTask Inputs/P00_PneumaticValves.IABPneumaticPI641_N11DigitalInput <-> 1. TxPDO/P00_PneumaticValves.IABPneumaticPI_N11DigitalInput
//     PlcTask Inputs/P00_PneumaticValves.IABPneumaticPI641_N12DigitalInput <-> 1. TxPDO/P00_PneumaticValves.IABPneumaticPI_N12DigitalInput
//     PlcTask Inputs/P00_PneumaticValves.IABPneumaticPI641_N13DigitalInput <-> 1. TxPDO/8 Digital Input 17-24
//     PlcTask Outputs/P00_PneumaticValves.QABPneumaticPI641ValveCoils[1] <-> 1. RxPDO/P00_PneumaticValves.QABPneumaticPI641ValveCoils[1]
//     PlcTask Outputs/P00_PneumaticValves.QABPneumaticPI641ValveCoils[2] <-> 1. RxPDO/P00_PneumaticValves.QABPneumaticPI641ValveCoils[2]
//     PlcTask Outputs/P00_PneumaticValves.QABPneumaticPI641ValveCoils[3] <-> 1. RxPDO/P00_PneumaticValves.QABPneumaticPI641ValveCoils[3]
//     PlcTask Outputs/P00_PneumaticValves.QABPneumaticPI641ValveCoils[4] <-> 1. RxPDO/Valve coils 25-32
//     PlcTask Outputs/P00_PneumaticValves.QABPneumaticPI641ValveCoils[5] <-> 1. RxPDO/Valve coils 33-40
//     PlcTask Outputs/P00_PneumaticValves.QABPneumaticPI641ValveCoils[6] <-> 1. RxPDO/Valve coils 41-48
//   (this object) <-> Device 1 (EtherCAT)/R2_242A1 (CU1128)/R2_242A1 (CU1128-C)/PI_71U2_TransDoKar (FR-E800-E)
//     PlcTask Inputs/P01_PucksInserter.uiPucksInserterConveyorActualVelocity <-> 1st Transmit PDO Mapping/Index:Pr.1330,Sub:Pr.1394(Low)
//     PlcTask Inputs/P01_PucksInserter.uiPucksInserterConveyorSW <-> 1st Transmit PDO Mapping/Statusword
//     PlcTask Outputs/P01_PucksInserter.udiPucksInserterConveyorVelocity <-> 1st Receive PDO Mapping/Index:Pr.1320,Sub:Pr.1389(Low)
//     PlcTask Outputs/P01_PucksInserter.uiPucksInserterConveyorCW <-> 1st Receive PDO Mapping/Controlword
//   (this object) <-> Device 1 (EtherCAT)/R2_242A1 (CU1128)/R2_242A1 (CU1128-C)/PI_71U3_StolPod (FR-E800-E)
//     PlcTask Inputs/P01_PucksInserter.InPucksInserterPushTable_m1_STW <-> Transmit PDO Mapping/Statusword
//     PlcTask Inputs/P01_PucksInserter.InPucksInserterPushTable_m1_VelocityCV <-> Transmit PDO Mapping/Pr.1330 Mapping
//     PlcTask Outputs/P01_PucksInserter.QnPucksInserterPushTable_m1_CTW <-> Receive PDO Mapping/Controlword
//     PlcTask Outputs/P01_PucksInserter.QnPucksInserterPushTable_m1_VelocitySV <-> Receive PDO Mapping/Pr.1320 Mapping
//   (this object) <-> Device 1 (EtherCAT)/R2_242A1 (CU1128)/R2_242A1 (CU1128-C)/PI_71U5_Rolka (FR-E800-E)
//     PlcTask Inputs/P01_PucksInserter.InPucksInserterPushTable_m2_STW <-> 1st Transmit PDO Mapping/Statusword
//     PlcTask Inputs/P01_PucksInserter.InPucksInserterPushTable_m2_VelocityCV <-> 1st Transmit PDO Mapping/Index:Pr.1330,Sub:Pr.1394(Low)
//     PlcTask Outputs/P01_PucksInserter.QnPucksInserterPushTable_m2_CTW <-> 1st Receive PDO Mapping/Controlword
//     PlcTask Outputs/P01_PucksInserter.QnPucksInserterPushTable_m2_VelocitySV <-> 1st Receive PDO Mapping/Index:Pr.1320,Sub:Pr.1389(Low)
//   (this object) <-> Device 1 (EtherCAT)/R2_242A1 (CU1128)/R2_242A1 (CU1128-C)/PI_71U6_DodatTor (FR-E800-E)
//     PlcTask Inputs/P01_PucksInserter.InPucksInserterPushTable_m3_STW <-> 1st Transmit PDO Mapping/Statusword
//     PlcTask Inputs/P01_PucksInserter.InPucksInserterPushTable_m3_VelocityCV <-> 1st Transmit PDO Mapping/Index:Pr.1330,Sub:Pr.1394(Low)
//     PlcTask Outputs/P01_PucksInserter.QnPucksInserterPushTable_m3_CTW <-> 1st Receive PDO Mapping/Controlword
//     PlcTask Outputs/P01_PucksInserter.QnPucksInserterPushTable_m3_VelocitySV <-> 1st Receive PDO Mapping/Index:Pr.1320,Sub:Pr.1389(Low)
//   (this object) <-> Device 1 (EtherCAT)/R2_242A1 (CU1128)/R2_242A1 (CU1128-C)/PI_BC4 (EK1914)
//     PlcTask Inputs/P01_PucksInserter.IbPucksInserterFuseDrivesOK <-> Module 2 (DIO)/DIO Inputs/Input 0
//     PlcTask Inputs/P01_PucksInserter.IbPucksInserterFuseFB1OK <-> Module 2 (DIO)/DIO Inputs/Input 3
//     PlcTask Inputs/P01_PucksInserter.IbPucksInserterTransporter1OK <-> Module 2 (DIO)/DIO Inputs/Input 1
//     PlcTask Inputs/P01_PucksInserter.IbPucksInserterTransporter2OK <-> Module 2 (DIO)/DIO Inputs/Input 2
//     PlcTask Outputs/GVL_IO.QbPickInserterDoorsClose <-> Module 2 (DIO)/DIO Outputs/Output 2
//     PlcTask Outputs/P01_PucksInserter.QbPucksInserterHammerHeightDownCmd <-> Module 2 (DIO)/DIO Outputs/Output 0
//     PlcTask Outputs/P01_PucksInserter.QbPucksInserterHammerHeightUpCmd <-> Module 2 (DIO)/DIO Outputs/Output 1
//   (this object) <-> Device 1 (EtherCAT)/R2_242A1 (CU1128)/R2_242A1 (CU1128-C)/PI_BC4 (EK1914)/PI_AI7 (EL5122)
//     PlcTask Inputs/P01_PucksInserter.IbPucksInserterHammerHeightEncoderSetCDone <-> ENC Status Channel 1/Status/Set counter done
//     PlcTask Inputs/P01_PucksInserter.IudiPucksInserterHammerHeightEncoderCV <-> ENC Status Channel 1/Counter value
//     PlcTask Outputs/P01_PucksInserter.QbPucksInserterHammerHeightEncoderSetC <-> ENC Control Channel 1/Control/Set counter
//     PlcTask Outputs/P01_PucksInserter.QudiPucksInserterHammerHeightEncoderSetCV <-> ENC Control Channel 1/Set counter value
//   (this object) <-> Device 1 (EtherCAT)/R2_242A1 (CU1128)/R2_242A1 (CU1128-C)/PI_BC4 (EK1914)/PI_DI5 (EL1008)
//     PlcTask Inputs/GVL_IO.IbEmergencyStopButtonPushtable2 <-> Channel 2/Input
//     PlcTask Inputs/GVL_IO.IbPucksInserterCycleStartButton <-> Channel 6/Input
//     PlcTask Inputs/GVL_IO.IbPucksInserterCycleStopButton <-> Channel 5/Input
//     PlcTask Inputs/GVL_IO.IbPucksInserterDoorsOpen <-> Channel 1/Input
//     PlcTask Inputs/GVL_IO.IbPucksInserterEmergencyStopButton0Pressed <-> Channel 3/Input
//     PlcTask Inputs/GVL_IO.IbPucksInserterEmergencyStopButton1Pressed <-> Channel 4/Input
//     PlcTask Inputs/GVL_IO.IbPucksInserterRollerFuse <-> Channel 8/Input
//     PlcTask Inputs/GVL_IO_SAFETY.bPucksInserterSafetyResetIn <-> Channel 7/GVL_IO.IbPI_SafetyResetIn
//   (this object) <-> Device 1 (EtherCAT)/R2_242A1 (CU1128)/R2_242A1 (CU1128-C)/PI_BC4 (EK1914)/PI_DO4 (EL2008)
//     PlcTask Outputs/P00_Signalization.QbPucksInserterResetLamp <-> Channel 2/Output
//     PlcTask Outputs/P00_Signalization.QbPucksInserterStartLamp <-> Channel 1/Output
//   (this object) <-> Device 1 (EtherCAT)/R2_242A1 (CU1128)/R2_242A1 (CU1128-C)/zew_616U1_Odrz (FR-E800-E)
//     PlcTask Inputs/P14_BadBottleConyevor.InBadBottleConveyorSTW <-> 1st Transmit PDO Mapping/Statusword
//     PlcTask Inputs/P14_BadBottleConyevor.InBadBottleConveyorVelocityCV <-> 1st Transmit PDO Mapping/Index:Pr.1330,Sub:Pr.1394(Low)
//     PlcTask Outputs/P14_BadBottleConyevor.QnBadBottleConveyorConvCTW <-> 1st Receive PDO Mapping/Controlword
//     PlcTask Outputs/P14_BadBottleConyevor.QnBadBottleConveyorVelocitySV <-> 1st Receive PDO Mapping/Index:Pr.1320,Sub:Pr.1389(Low)
//   (this object) <-> Device 1 (EtherCAT)/R2_242A1 (CU1128)/R2_242A1 (CU1128-C)/zew_617U1_Wyj 126 (FR-E800-E)
//     PlcTask Inputs/P17_TurnTables.InExitConveyorSTW <-> 1st Transmit PDO Mapping/Statusword
//     PlcTask Inputs/P17_TurnTables.InExitConveyorVelocityCV <-> 1st Transmit PDO Mapping/Index:Pr.1330,Sub:Pr.1394(Low)
//     PlcTask Outputs/P17_TurnTables.QnExitConveyorConvCTW <-> 1st Receive PDO Mapping/Controlword
//     PlcTask Outputs/P17_TurnTables.QnExitConveyorVelocitySV <-> 1st Receive PDO Mapping/Index:Pr.1320,Sub:Pr.1389(Low)
//   (this object) <-> Device 1 (EtherCAT)/R2_646N1 (EtherCAT EB80 series)
//     PlcTask Inputs/P00_PneumaticValves.IABPneumatic646_N11DigitalInput <-> 1. TxPDO/8 Digital Input 1-8
//     PlcTask Inputs/P00_PneumaticValves.IABPneumatic646_N12DigitalInput <-> 1. TxPDO/8 Digital Input 9-16
//     PlcTask Inputs/P00_PneumaticValves.IABPneumatic646_N13DigitalInput <-> 1. TxPDO/8 Digital Input 17-24
//     PlcTask Outputs/P00_PneumaticValves.QABPneumatic646ValveCoils[1] <-> 1. RxPDO/Valve coils 1-8
//     PlcTask Outputs/P00_PneumaticValves.QABPneumatic646ValveCoils[2] <-> 1. RxPDO/Valve coils 9-16
//     PlcTask Outputs/P00_PneumaticValves.QABPneumatic646ValveCoils[3] <-> 1. RxPDO/Valve coils 17-24
//     PlcTask Outputs/P00_PneumaticValves.QABPneumatic646ValveCoils[4] <-> 1. RxPDO/Valve coils 25-32
//     PlcTask Outputs/P00_PneumaticValves.QABPneumatic646ValveCoils[5] <-> 1. RxPDO/Valve coils 33-40
//   (this object) <-> Device 1 (EtherCAT)/R2_BC1 (EK1100)/AI1 (EL3356-0010)
//     WeightTask Inputs/P05_Weight.IbWeight1CalibrationInProgress <-> RMB Status/Status/Calibration in progress
//     WeightTask Inputs/P05_Weight.IbWeight1DataInvalid <-> RMB Status/Status/Data invalid
//     WeightTask Inputs/P05_Weight.IbWeight1Error <-> RMB Status/Status/Error
//     WeightTask Inputs/P05_Weight.IbWeight1Overrange <-> RMB Status/Status/Overrange
//     WeightTask Inputs/P05_Weight.IbWeight1SteadyState <-> RMB Status/Status/Steady state
//     WeightTask Inputs/P05_Weight.IbWeight1SyncError <-> RMB Status/Status/Sync error
//     WeightTask Inputs/P05_Weight.InWeight1Value <-> RMB Value (INT32)/Value
//     WeightTask Outputs/P05_Weight.QbWeight1DisableCalibration <-> RMB Control/Ctrl/Disable calibration
//     WeightTask Outputs/P05_Weight.QbWeight1InputFreeze <-> RMB Control/Ctrl/Input freeze
//     WeightTask Outputs/P05_Weight.QbWeight1SampleMode <-> RMB Control/Ctrl/Sample mode
//     WeightTask Outputs/P05_Weight.QbWeight1StartCalibration <-> RMB Control/Ctrl/Start calibration
//     WeightTask Outputs/P05_Weight.QbWeight1Tara <-> RMB Control/Ctrl/Tara
//   (this object) <-> Device 1 (EtherCAT)/R2_BC1 (EK1100)/AI2 (EL3356-0010)
//     WeightTask Inputs/P05_Weight.IbWeight2CalibrationInProgress <-> RMB Status/Status/Calibration in progress
//     WeightTask Inputs/P05_Weight.IbWeight2DataInvalid <-> RMB Status/Status/Data invalid
//     WeightTask Inputs/P05_Weight.IbWeight2Error <-> RMB Status/Status/Error
//     WeightTask Inputs/P05_Weight.IbWeight2Overrange <-> RMB Status/Status/Overrange
//     WeightTask Inputs/P05_Weight.IbWeight2SteadyState <-> RMB Status/Status/Steady state
//     WeightTask Inputs/P05_Weight.IbWeight2SyncError <-> RMB Status/Status/Sync error
//     WeightTask Inputs/P05_Weight.InWeight2Value <-> RMB Value (INT32)/Value
//     WeightTask Outputs/P05_Weight.QbWeight2DisableCalibration <-> RMB Control/Ctrl/Disable calibration
//     WeightTask Outputs/P05_Weight.QbWeight2InputFreeze <-> RMB Control/Ctrl/Input freeze
//     WeightTask Outputs/P05_Weight.QbWeight2SampleMode <-> RMB Control/Ctrl/Sample mode
//     WeightTask Outputs/P05_Weight.QbWeight2StartCalibration <-> RMB Control/Ctrl/Start calibration
//     WeightTask Outputs/P05_Weight.QbWeight2Tara <-> RMB Control/Ctrl/Tara
//   (this object) <-> Device 1 (EtherCAT)/R2_BC1 (EK1100)/AI3 (EL3356-0010)
//     WeightTask Inputs/P05_Weight.IbWeight3CalibrationInProgress <-> RMB Status/Status/Calibration in progress
//     WeightTask Inputs/P05_Weight.IbWeight3DataInvalid <-> RMB Status/Status/Data invalid
//     WeightTask Inputs/P05_Weight.IbWeight3Error <-> RMB Status/Status/Error
//     WeightTask Inputs/P05_Weight.IbWeight3Overrange <-> RMB Status/Status/Overrange
//     WeightTask Inputs/P05_Weight.IbWeight3SteadyState <-> RMB Status/Status/Steady state
//     WeightTask Inputs/P05_Weight.IbWeight3SyncError <-> RMB Status/Status/Sync error
//     WeightTask Inputs/P05_Weight.InWeight3Value <-> RMB Value (INT32)/Value
//     WeightTask Outputs/P05_Weight.QbWeight3DisableCalibration <-> RMB Control/Ctrl/Disable calibration
//     WeightTask Outputs/P05_Weight.QbWeight3InputFreeze <-> RMB Control/Ctrl/Input freeze
//     WeightTask Outputs/P05_Weight.QbWeight3SampleMode <-> RMB Control/Ctrl/Sample mode
//     WeightTask Outputs/P05_Weight.QbWeight3StartCalibration <-> RMB Control/Ctrl/Start calibration
//     WeightTask Outputs/P05_Weight.QbWeight3Tara <-> RMB Control/Ctrl/Tara
//   (this object) <-> Device 1 (EtherCAT)/R2_BC1 (EK1100)/AI4 (EL3356-0010)
//     WeightTask Inputs/P05_Weight.IbWeight4CalibrationInProgress <-> RMB Status/Status/Calibration in progress
//     WeightTask Inputs/P05_Weight.IbWeight4DataInvalid <-> RMB Status/Status/Data invalid
//     WeightTask Inputs/P05_Weight.IbWeight4Error <-> RMB Status/Status/Error
//     WeightTask Inputs/P05_Weight.IbWeight4Overrange <-> RMB Status/Status/Overrange
//     WeightTask Inputs/P05_Weight.IbWeight4SteadyState <-> RMB Status/Status/Steady state
//     WeightTask Inputs/P05_Weight.IbWeight4SyncError <-> RMB Status/Status/Sync error
//     WeightTask Inputs/P05_Weight.InWeight4Value <-> RMB Value (INT32)/Value
//     WeightTask Outputs/P05_Weight.QbWeight4DisableCalibration <-> RMB Control/Ctrl/Disable calibration
//     WeightTask Outputs/P05_Weight.QbWeight4InputFreeze <-> RMB Control/Ctrl/Input freeze
//     WeightTask Outputs/P05_Weight.QbWeight4SampleMode <-> RMB Control/Ctrl/Sample mode
//     WeightTask Outputs/P05_Weight.QbWeight4StartCalibration <-> RMB Control/Ctrl/Start calibration
//     WeightTask Outputs/P05_Weight.QbWeight4Tara <-> RMB Control/Ctrl/Tara
//   (this object) <-> Device 1 (EtherCAT)/R2_BC1 (EK1100)/AI5 (EL3356-0010)
//     WeightTask Inputs/P05_Weight.IbWeight5CalibrationInProgress <-> RMB Status/Status/Calibration in progress
//     WeightTask Inputs/P05_Weight.IbWeight5DataInvalid <-> RMB Status/Status/Data invalid
//     WeightTask Inputs/P05_Weight.IbWeight5Error <-> RMB Status/Status/Error
//     WeightTask Inputs/P05_Weight.IbWeight5Overrange <-> RMB Status/Status/Overrange
//     WeightTask Inputs/P05_Weight.IbWeight5SteadyState <-> RMB Status/Status/Steady state
//     WeightTask Inputs/P05_Weight.IbWeight5SyncError <-> RMB Status/Status/Sync error
//     WeightTask Inputs/P05_Weight.InWeight5Value <-> RMB Value (INT32)/Value
//     WeightTask Outputs/P05_Weight.QbWeight5DisableCalibration <-> RMB Control/Ctrl/Disable calibration
//     WeightTask Outputs/P05_Weight.QbWeight5InputFreeze <-> RMB Control/Ctrl/Input freeze
//     WeightTask Outputs/P05_Weight.QbWeight5SampleMode <-> RMB Control/Ctrl/Sample mode
//     WeightTask Outputs/P05_Weight.QbWeight5StartCalibration <-> RMB Control/Ctrl/Start calibration
//     WeightTask Outputs/P05_Weight.QbWeight5Tara <-> RMB Control/Ctrl/Tara
//   (this object) <-> Device 1 (EtherCAT)/R2_BC1 (EK1100)/AI6 (EL3356-0010)
//     WeightTask Inputs/P05_Weight.IbWeight6CalibrationInProgress <-> RMB Status/Status/Calibration in progress
//     WeightTask Inputs/P05_Weight.IbWeight6DataInvalid <-> RMB Status/Status/Data invalid
//     WeightTask Inputs/P05_Weight.IbWeight6Error <-> RMB Status/Status/Error
//     WeightTask Inputs/P05_Weight.IbWeight6Overrange <-> RMB Status/Status/Overrange
//     WeightTask Inputs/P05_Weight.IbWeight6SteadyState <-> RMB Status/Status/Steady state
//     WeightTask Inputs/P05_Weight.IbWeight6SyncError <-> RMB Status/Status/Sync error
//     WeightTask Inputs/P05_Weight.InWeight6Value <-> RMB Value (INT32)/Value
//     WeightTask Outputs/P05_Weight.QbWeight6DisableCalibration <-> RMB Control/Ctrl/Disable calibration
//     WeightTask Outputs/P05_Weight.QbWeight6InputFreeze <-> RMB Control/Ctrl/Input freeze
//     WeightTask Outputs/P05_Weight.QbWeight6SampleMode <-> RMB Control/Ctrl/Sample mode
//     WeightTask Outputs/P05_Weight.QbWeight6StartCalibration <-> RMB Control/Ctrl/Start calibration
//     WeightTask Outputs/P05_Weight.QbWeight6Tara <-> RMB Control/Ctrl/Tara
//   (this object) <-> Device 1 (EtherCAT)/R2_BC1 (EK1100)/AI7 (EL5122)
//     PlcTask Inputs/P02_Dispencers.IbDispencersCatchHeightEncoderSetCDone <-> ENC Status Channel 1/Status/Set counter done
//     PlcTask Inputs/P02_Dispencers.IudiDispencersCatchHeightEncoderCV <-> ENC Status Channel 1/Counter value
//     PlcTask Inputs/P09_CapPuttedCheck.IbCapPuttedCheckEncoderSetCDone <-> ENC Status Channel 2/Status/Set counter done
//     PlcTask Inputs/P09_CapPuttedCheck.IudiCapPuttedCheckHeightEncoderCV <-> ENC Status Channel 2/Counter value
//     PlcTask Outputs/P02_Dispencers.QbDispencersCatchHeightEncoderSetC <-> ENC Control Channel 1/Control/Set counter
//     PlcTask Outputs/P02_Dispencers.QudiDispencersCatchHeightEncoderSetCV <-> ENC Control Channel 1/Set counter value
//     PlcTask Outputs/P09_CapPuttedCheck.QbCapPuttedCheckHeightEncoderSetC <-> ENC Control Channel 2/Control/Set counter
//     PlcTask Outputs/P09_CapPuttedCheck.QudiCapPuttedCheckHeightEncoderSetCV <-> ENC Control Channel 2/Set counter value
//   (this object) <-> Device 1 (EtherCAT)/R2_BC1 (EK1100)/AI8 (EL5122)
//     PlcTask Inputs/P10_GripperScrewer.IbGripperScrewersHeightEncoderSetCDone <-> ENC Status Channel 1/Status/Set counter done
//     PlcTask Inputs/P10_GripperScrewer.IudiGripperScrewersHeightEncoderCV <-> ENC Status Channel 1/Counter value
//     PlcTask Inputs/P11_CapCorrectCheck.IbCapCorrectCheckEncoderSetCDone <-> ENC Status Channel 2/Status/Set counter done
//     PlcTask Inputs/P11_CapCorrectCheck.IudiCapCorrectCheckHeightEncoderCV <-> ENC Status Channel 2/Counter value
//     PlcTask Outputs/P10_GripperScrewer.QbGripperScrewersHeightEncoderSetC <-> ENC Control Channel 1/Control/Set counter
//     PlcTask Outputs/P10_GripperScrewer.QudiGripperScrewersHeightEncoderSetCV <-> ENC Control Channel 1/Set counter value
//     PlcTask Outputs/P11_CapCorrectCheck.QbCapCorrectCheckHeightEncoderSetC <-> ENC Control Channel 2/Control/Set counter
//     PlcTask Outputs/P11_CapCorrectCheck.QudiCapCorrectCheckHeightEncoderSetCV <-> ENC Control Channel 2/Set counter value
//   (this object) <-> Device 1 (EtherCAT)/R2_BC1 (EK1100)/AI9 (EL5122)
//     PlcTask Inputs/P06_WickFeeder.IbWickFeederHeightEncoderSetCDone <-> ENC Status Channel 1/Status/Set counter done
//     PlcTask Inputs/P06_WickFeeder.IudiWickFeederHeightEncoderCV <-> ENC Status Channel 1/Counter value
//     PlcTask Outputs/P06_WickFeeder.QbWickFeederHeightEncoderSetC <-> ENC Control Channel 1/Control/Set counter
//     PlcTask Outputs/P06_WickFeeder.QudiWickFeederHeightEncoderSetCV <-> ENC Control Channel 1/Set counter value
//   (this object) <-> Device 1 (EtherCAT)/R2_BC1 (EK1100)/DI1 (EL1809)
//     PlcTask Inputs/GVL_IO.IbCompressedAirOK <-> Channel 13/GVL_IO.IbCompressedAirOK
//     PlcTask Inputs/GVL_IO.IbCycleStartButton <-> Channel 14/GVL_IO.IbCycleStartButton
//     PlcTask Inputs/GVL_IO.IbCycleStopButton <-> Channel 16/GVL_IO.IbCycleStopButton
//     PlcTask Inputs/GVL_IO.IbDCSupply1OK <-> Channel 2/GVL_IO.IbDCSupply1OK
//     PlcTask Inputs/GVL_IO.IbDCSupply2OK <-> Channel 3/GVL_IO.IbDCSupply2OK
//     PlcTask Inputs/GVL_IO.IbDCSupply3OK <-> Channel 4/GVL_IO.IbDCSupply3OK
//     PlcTask Inputs/GVL_IO.IbFuseDrivesOK <-> Channel 8/GVL_IO.IbFuseDrivesOK
//     PlcTask Inputs/GVL_IO.IbFuseFB1OK <-> Channel 5/GVL_IO.IbFuseFB1OK
//     PlcTask Inputs/GVL_IO.IbFuseFB2OK <-> Channel 6/GVL_IO.IbFuseFB2OK
//     PlcTask Inputs/GVL_IO.IbPowerSupplyOK <-> Channel 1/GVL_IO.IbPowerSupplyOK
//     PlcTask Inputs/GVL_IO_SAFETY.IbSafetyRelayJiecang <-> Channel 9/GVL_IO_SAFETY.IbSafetyRelayJiecang
//     PlcTask Inputs/GVL_IO_SAFETY.IbSafetyRelayMotorsRobotA <-> Channel 11/GVL_IO.IbCompressedAirOK
//     PlcTask Inputs/GVL_IO_SAFETY.IbSafetyRelayMotorsRobotB <-> Channel 12/GVL_IO.IbCycleStartButton
//     PlcTask Inputs/GVL_IO_SAFETY.IbSafetyRelayPneumatics <-> Channel 10/GVL_IO_SAFETY.IbSafetyRelaySteppers
//     PlcTask Inputs/GVL_IO_SAFETY.bSafetyResetIn <-> Channel 15/GVL_IO_SAFETY.bSafetyResetIn
//   (this object) <-> Device 1 (EtherCAT)/R2_BC1 (EK1100)/DI2 (EL1809)
//     PlcTask Inputs/GVL_IO.IbBottleTransferDoorsOpen <-> Channel 10/GVL_IO.IbBottleTransferDoorsOpen
//     PlcTask Inputs/GVL_IO.IbDispencersDoorsOpen <-> Channel 6/GVL_IO.IbDispencersDoorsOpen
//     PlcTask Inputs/GVL_IO.IbEmergencyStopButton0Pressed <-> Channel 1/GVL_IO.IbEmergencyStopButton0Pressed
//     PlcTask Inputs/GVL_IO.IbEmergencyStopButton1Pressed <-> Channel 3/GVL_IO.IbEmergencyStopButton1Pressed
//     PlcTask Inputs/GVL_IO.IbEmergencyStopButton2Pressed <-> Channel 5/GVL_IO.IbEmergencyStopButton2Pressed
//     PlcTask Inputs/GVL_IO.IbEmergencyStopButton3Pressed <-> Channel 4/GVL_IO.IbEmergencyStopButton3Pressed
//     PlcTask Inputs/GVL_IO.IbEmergencyStopButton4Pressed <-> Channel 2/GVL_IO.IbEmergencyStopButton4Pressed
//     PlcTask Inputs/GVL_IO.IbGripperScrewerDoorsOpen <-> Channel 8/GVL_IO.IbGripperScrewerDoorsOpen
//     PlcTask Inputs/GVL_IO.IbLidSealingDoorsOpen <-> Channel 7/GVL_IO.IbLidSealingDoorsOpen
//     PlcTask Inputs/GVL_IO.IbTanksDoorsOpen <-> Channel 9/GVL_IO.IbTanksDoorsOpen
//     PlcTask Inputs/P02_Dispencers.IbTank1PumpFuseOK <-> Channel 11/P02_Dispencers.IbTank1PumpFuseOK
//     PlcTask Inputs/P02_Dispencers.IbTank2PumpFuseOK <-> Channel 12/P02_Dispencers.IbTank2PumpFuseOK
//     PlcTask Inputs/P02_Dispencers.IbTank3PumpFuseOK <-> Channel 13/P02_Dispencers.IbTank3PumpFuseOK
//     PlcTask Inputs/P02_Dispencers.IbTank4PumpFuseOK <-> Channel 14/P02_Dispencers.IbTank4PumpFuseOK
//     PlcTask Inputs/P16_LabelMachine.IbLabelMachineNotError <-> Channel 16/P16_LabelMachine.IbLabelMachineNotError
//     PlcTask Inputs/P16_LabelMachine.IbLabelMachineWorking <-> Channel 15/P16_LabelMachine.IbLabelMachineWorking
//   (this object) <-> Device 1 (EtherCAT)/R2_BC1 (EK1100)/DO1 (EL2809)
//     PlcTask Outputs/GVL_IO.QbBottleTransferDoorsClose <-> Channel 8/GVL_IO.QbBottleTransferDoorsClose
//     PlcTask Outputs/GVL_IO.QbDispencersDoorsClose <-> Channel 4/GVL_IO.QbDispencersDoorsClose
//     PlcTask Outputs/GVL_IO.QbGripperScrewerClose <-> Channel 6/GVL_IO.QbGripperScrewerClose
//     PlcTask Outputs/GVL_IO.QbLidSealingDoorsClose <-> Channel 5/GVL_IO.QbLidSealingDoorsClose
//     PlcTask Outputs/GVL_IO.QbResetFuseFB1 <-> Channel 1/GVL_IO.QbResetFuseFB1
//     PlcTask Outputs/GVL_IO.QbResetFuseFB2 <-> Channel 2/GVL_IO.QbResetFuseFB2
//     PlcTask Outputs/GVL_IO.QbTanksDoorsClose <-> Channel 7/GVL_IO.QbTanksDoorsClose
//     PlcTask Outputs/P00_Signalization.QbBuzzer <-> Channel 13/P00_Signalization.QbBuzzer
//     PlcTask Outputs/P00_Signalization.QbResetLamp <-> Channel 12/P00_Signalization.QbResetLamp
//     PlcTask Outputs/P00_Signalization.QbStartLamp <-> Channel 11/P00_Signalization.QbStartLamp
//     PlcTask Outputs/P13_BottleTransfer.QbBottleTransferRobotMode1 <-> Channel 9/P13_BottleTransfer.QbBottleTransferRobotMode1
//     PlcTask Outputs/P13_BottleTransfer.QbBottleTransferRobotMode2 <-> Channel 10/P13_BottleTransfer.QbBottleTransferRobotMode2
//   (this object) <-> Device 1 (EtherCAT)/R2_BC1 (EK1100)/DO2 (EL2809)
//     PlcTask Outputs/P02_Dispencers.QbDispencersCatch1HeightDownCmd <-> Channel 2/P02_Dispencers.QbDispencersCatch1HeightDownCmd
//     PlcTask Outputs/P02_Dispencers.QbDispencersCatch1HeightUpCmd <-> Channel 1/P02_Dispencers.QbDispencersCatch1HeightUpCmd
//     PlcTask Outputs/P02_Dispencers.QbTank1PumpStart <-> Channel 11/Rezerwa
//     PlcTask Outputs/P02_Dispencers.QbTank2PumpStart <-> Channel 12/Rezerwa
//     PlcTask Outputs/P02_Dispencers.QbTank3PumpStart <-> Channel 13/P02_Dispencers.QbTank1PumpStart
//     PlcTask Outputs/P02_Dispencers.QbTank4PumpStart <-> Channel 14/P02_Dispencers.QbTank2PumpStart
//     PlcTask Outputs/P10_GripperScrewer.QbGripperScrewer1CatchHeightDownCmd <-> Channel 5/P10_GripperScrewer.QbGripperScrewer1CatchHeightDownCmd
//     PlcTask Outputs/P10_GripperScrewer.QbGripperScrewer1CatchHeightUpCmd <-> Channel 6/P10_GripperScrewer.QbGripperScrewer1CatchHeightUpCmd
//     PlcTask Outputs/P11_CapCorrectCheck.QbCapCorrectCheckHeightDownCmd <-> Channel 7/P11_CapCorrectCheck.QbCapCorrectCheckHeightDownCmd
//     PlcTask Outputs/P11_CapCorrectCheck.QbCapCorrectCheckHeightUpCmd <-> Channel 8/P11_CapCorrectCheck.QbCapCorrectCheckHeightUpCmd
//     PlcTask Outputs/P16_LabelMachine.QbLabelMachineStart <-> Channel 15/P16_LabelMachine.QbLabelMachineStart
//     PlcTask Outputs/P16_LabelMachine.QbLabelMachineStop <-> Channel 16/P16_LabelMachine.QbLabelMachineStop
//   (this object) <-> Device 1 (EtherCAT)/R2_BC1 (EK1100)/DO3 (EL2809)
//     PlcTask Outputs/P06_WickFeeder.QbWickFeeder_HeightMotorDown <-> Channel 1/P06_WickFeeder.QbWickFeeder_HeightMotorUp
//     PlcTask Outputs/P06_WickFeeder.QbWickFeeder_HeightMotorUp <-> Channel 2/P06_WickFeeder.QbWickFeeder_HeightMotorDown
//   (this object) <-> Device 1 (EtherCAT)/R2_BC1 (EK1100)/DO4 (EL2564)
//     PlcTask Outputs/P00_Signalization.QiLineBlueSignalizationLamp <-> PWM Outputs Channel 3/BLUE PWM output
//     PlcTask Outputs/P00_Signalization.QiLineGreenSignalizationLamp <-> PWM Outputs Channel 2/GREEN PWM output
//     PlcTask Outputs/P00_Signalization.QiLineRedSignalizationLamp <-> PWM Outputs Channel 1/RED PWM output
//     PlcTask Outputs/P00_Signalization.QiLineWhiteSignalizationLamp <-> PWM Outputs Channel 4/WHITE PWM output
//   (this object) <-> Device 1 (EtherCAT)/R2_BC1 (EK1100)/SI2 (EL1918)
//     PlcTask Inputs/GVL_IO.IbBottleSorterDisable <-> Module 1 (FSOE)/FSoE Inputs/FSOE/FSIN Module 3.Input
//     PlcTask Inputs/GVL_IO.IbCapSorterDisable <-> Module 1 (FSOE)/FSoE Inputs/FSOE/FSIN Module 1.Input
//   (this object) <-> NC-Task 1 SAF/Axes/Doz1
//     PlcTask Inputs/GVL.aDispencer1AxisRef.NcToPlc <-> Outputs/ToPlc
//     PlcTask Outputs/GVL.aDispencer1AxisRef.PlcToNc <-> Inputs/FromPlc
//   (this object) <-> NC-Task 1 SAF/Axes/Doz2
//     PlcTask Inputs/GVL.aDispencer2AxisRef.NcToPlc <-> Outputs/ToPlc
//     PlcTask Outputs/GVL.aDispencer2AxisRef.PlcToNc <-> Inputs/FromPlc
//   (this object) <-> NC-Task 1 SAF/Axes/Doz3
//     PlcTask Inputs/GVL.aDispencer3AxisRef.NcToPlc <-> Outputs/ToPlc
//     PlcTask Outputs/GVL.aDispencer3AxisRef.PlcToNc <-> Inputs/FromPlc
//   (this object) <-> NC-Task 1 SAF/Axes/Doz4
//     PlcTask Inputs/GVL.aDispencer4AxisRef.NcToPlc <-> Outputs/ToPlc
//     PlcTask Outputs/GVL.aDispencer4AxisRef.PlcToNc <-> Inputs/FromPlc
//   (this object) <-> NC-Task 1 SAF/Axes/PI_Karusela
//     PlcTask Inputs/GVL.aPucksInserterWheelAxisRef.NcToPlc <-> Outputs/ToPlc
//     PlcTask Outputs/GVL.aPucksInserterWheelAxisRef.PlcToNc <-> Inputs/FromPlc
//   (this object) <-> NC-Task 1 SAF/Axes/PodDoz12
//     PlcTask Inputs/GVL.aDispencerLifter12AxisRef.NcToPlc <-> Outputs/ToPlc
//     PlcTask Outputs/GVL.aDispencerLifter12AxisRef.PlcToNc <-> Inputs/FromPlc
//   (this object) <-> NC-Task 1 SAF/Axes/PodDoz34
//     PlcTask Inputs/GVL.aDispencerLifter34AxisRef.NcToPlc <-> Outputs/ToPlc
//     PlcTask Outputs/GVL.aDispencerLifter34AxisRef.PlcToNc <-> Inputs/FromPlc
//   (this object) <-> NC-Task 1 SAF/Axes/PodZak1
//     PlcTask Inputs/GVL.aGripperScrewer1LiftAxisRef.NcToPlc <-> Outputs/ToPlc
//     PlcTask Outputs/GVL.aGripperScrewer1LiftAxisRef.PlcToNc <-> Inputs/FromPlc
//   (this object) <-> NC-Task 1 SAF/Axes/PodZak2
//     PlcTask Inputs/GVL.aGripperScrewer2LiftAxisRef.NcToPlc <-> Outputs/ToPlc
//     PlcTask Outputs/GVL.aGripperScrewer2LiftAxisRef.PlcToNc <-> Inputs/FromPlc
//   (this object) <-> NC-Task 1 SAF/Axes/PrzecDoz
//     PlcTask Inputs/GVL.aFormsDragingLeftAxisRef.NcToPlc <-> Outputs/ToPlc
//     PlcTask Outputs/GVL.aFormsDragingLeftAxisRef.PlcToNc <-> Inputs/FromPlc
//   (this object) <-> NC-Task 1 SAF/Axes/PrzecDoz2
//     PlcTask Inputs/GVL.aFormsDragingRightAxisRef.NcToPlc <-> Outputs/ToPlc
//     PlcTask Outputs/GVL.aFormsDragingRightAxisRef.PlcToNc <-> Inputs/FromPlc
//   (this object) <-> NC-Task 1 SAF/Axes/PrzecGrz
//     PlcTask Inputs/GVL.aLidSealerDragingAxisRef.NcToPlc <-> Outputs/ToPlc
//     PlcTask Outputs/GVL.aLidSealerDragingAxisRef.PlcToNc <-> Inputs/FromPlc
//   (this object) <-> NC-Task 1 SAF/Axes/PrzecPlat
//     PlcTask Inputs/GVL.aWickFeederDragingAxisRef.NcToPlc <-> Outputs/ToPlc
//     PlcTask Outputs/GVL.aWickFeederDragingAxisRef.PlcToNc <-> Inputs/FromPlc
//   (this object) <-> NC-Task 1 SAF/Axes/PrzecSorNak
//     PlcTask Inputs/GVL.aCapSorterDragAxisRef.NcToPlc <-> Outputs/ToPlc
//     PlcTask Outputs/GVL.aCapSorterDragAxisRef.PlcToNc <-> Inputs/FromPlc
//   (this object) <-> NC-Task 1 SAF/Axes/PrzecZak
//     PlcTask Inputs/GVL.aBottleDragingAxisRef.NcToPlc <-> Outputs/ToPlc
//     PlcTask Outputs/GVL.aBottleDragingAxisRef.PlcToNc <-> Inputs/FromPlc
//   (this object) <-> NC-Task 1 SAF/Axes/VirtualDos
//     PlcTask Inputs/P02_DispencersCharts.DispencerAxisRef.NcToPlc <-> Outputs/ToPlc
//     PlcTask Outputs/P02_DispencersCharts.DispencerAxisRef.PlcToNc <-> Inputs/FromPlc
//   (this object) <-> NC-Task 1 SAF/Axes/VirtualPodDoz
//     PlcTask Inputs/P02_DispencersCharts.DispencerLifterAxisRef.NcToPlc <-> Outputs/ToPlc
//     PlcTask Outputs/P02_DispencersCharts.DispencerLifterAxisRef.PlcToNc <-> Inputs/FromPlc
//   (this object) <-> NC-Task 1 SAF/Axes/Zak1
//     PlcTask Inputs/GVL.aGripperScrewer1AxisRef.NcToPlc <-> Outputs/ToPlc
//     PlcTask Outputs/GVL.aGripperScrewer1AxisRef.PlcToNc <-> Inputs/FromPlc
//   (this object) <-> NC-Task 1 SAF/Axes/Zak2
//     PlcTask Inputs/GVL.aGripperScrewer2AxisRef.NcToPlc <-> Outputs/ToPlc
//     PlcTask Outputs/GVL.aGripperScrewer2AxisRef.PlcToNc <-> Inputs/FromPlc
//   (this object) <-> NC-Task 1 SAF/Axes/ZakEncoder1
//     PlcTask Inputs/GVL.aGripperScrewer1EncoderAxisRef.NcToPlc <-> Outputs/ToPlc
//     PlcTask Outputs/GVL.aGripperScrewer1EncoderAxisRef.PlcToNc <-> Inputs/FromPlc
//   (this object) <-> NC-Task 1 SAF/Axes/ZakEncoder2
//     PlcTask Inputs/GVL.aGripperScrewer2EncoderAxisRef.NcToPlc <-> Outputs/ToPlc
//     PlcTask Outputs/GVL.aGripperScrewer2EncoderAxisRef.PlcToNc <-> Inputs/FromPlc
//   (this object) <-> SafetyPLC/SafetyPLC Instance
//     PlcTask Inputs/GVL_IO.IbBottleFeederSafety <-> PlcTask Outputs/GVL_IO_SAFETY.QbBottleFeederSafety
//     PlcTask Inputs/GVL_IO.IbCommunicationErrorUF50 <-> PlcTask Outputs/GVL_IO_SAFETY.QbCommunicationErrorUF50
//     PlcTask Inputs/GVL_IO.IbCommunicationErrorUP50B <-> PlcTask Outputs/GVL_IO_SAFETY.QbCommunicationErrorUP50B
//     PlcTask Inputs/GVL_IO.IbEmergencyStopButton <-> PlcTask Outputs/GVL_IO_SAFETY.QbEmergencyStopButton
//     PlcTask Inputs/GVL_IO.IbSafetyResetIn <-> PlcTask Outputs/GVL_IO_SAFETY.bSafetyResetOut
//     PlcTask Outputs/GVL_IO.QbSafetyResetBottleSorterIn <-> PlcTask Inputs/GVL_IO_SAFETY.IbSafetyResetBottleSorterIn
//     PlcTask Outputs/GVL_IO.QbSafetyResetCapSorterIn <-> PlcTask Inputs/GVL_IO_SAFETY.IbSafetyResetCapSorterIn
//     PlcTask Outputs/GVL_IO.QbSafetyResetDelay <-> PlcTask Inputs/GVL_IO_SAFETY.IbSafetyResetDelay
//     WeightTask Inputs/GVL_IO.IbEmergencyStop <-> PlcTask Outputs/GVL_IO_SAFETY.QbEmergencyStop
//   (this object) <-> Device 1 (EtherCAT)/R2_242A1 (CU1128)/R2_242A1 (CU1128-B)/RC40_BC1(EK1814)
//     PlcTask Inputs/GVL_IO_SAFETY.bSafetyResetInRC40 <-> Channel 3/bSafetyResetInRC40
//   (this object) <-> Device 1 (EtherCAT)/R2_BC1 (EK1100)/CO2 (EL6910)
//     PlcTask Inputs/GVL_IO_SAFETY.IbComErr_Gr2 <-> StandardInputs/TwinSafeGroup2.ComErr_159
//     PlcTask Inputs/GVL_IO_SAFETY.IbComErr_Gr3 <-> StandardInputs/TwinSafeGroup3.ComErr_160
//     PlcTask Inputs/GVL_IO_SAFETY.IbFBErr_Gr2 <-> StandardInputs/TwinSafeGroup2.FBErr_156
//     PlcTask Inputs/GVL_IO_SAFETY.IbFBErr_Gr3 <-> StandardInputs/TwinSafeGroup3.FBErr_153
//     PlcTask Inputs/GVL_IO_SAFETY.IbOtherErr_Gr2 <-> StandardInputs/TwinSafeGroup2.OtherErr_157
//     PlcTask Inputs/GVL_IO_SAFETY.IbOtherErr_Gr3 <-> StandardInputs/TwinSafeGroup3.OtherErr_154
//     PlcTask Inputs/GVL_IO_SAFETY.IbOutErr_Gr2 <-> StandardInputs/TwinSafeGroup2.OutErr_158
//     PlcTask Inputs/GVL_IO_SAFETY.IbOutErr_Gr3 <-> StandardInputs/TwinSafeGroup3.OutErr_155
//     PlcTask Inputs/GVL_IO_SAFETY.IbUF50Deactivated <-> StandardInputs/TwinSafeGroup1.UF50_Deactivation_178
//     PlcTask Inputs/GVL_IO_SAFETY.IbUP50BDeactivated <-> StandardInputs/TwinSafeGroup1.UP50B_Deactivation_179
//     PlcTask Inputs/GVL_IO_SAFETY.bEmergencyStop <-> StandardInputs/TwinSafeGroup1.EStopStatus_44
//     PlcTask Inputs/GVL_IO_SAFETY.bEmergencyStopButton <-> StandardInputs/TwinSafeGroup1.EStopButton_43
//     PlcTask Outputs/GVL_IO_SAFETY.QbRUN_STOP <-> StandardOutputs/TwinSafeGroup1.Run_Stop_47
//     PlcTask Outputs/GVL_IO_SAFETY.QbRUN_STOP_GR2 <-> StandardOutputs/TwinSafeGroup2.Run_150
//     PlcTask Outputs/GVL_IO_SAFETY.QbRUN_STOP_GR3 <-> StandardOutputs/TwinSafeGroup3.Run_148
//     PlcTask Outputs/GVL_IO_SAFETY.bErrorAck <-> StandardOutputs/TwinSafeGroup1.ErrAck_42
//     PlcTask Outputs/GVL_IO_SAFETY.bErrorAckGr2 <-> StandardOutputs/TwinSafeGroup2.ErrAck_149
//     PlcTask Outputs/GVL_IO_SAFETY.bErrorAckGr3 <-> StandardOutputs/TwinSafeGroup3.ErrAck_147
//     PlcTask Outputs/GVL_IO_SAFETY.bSafetyReset <-> StandardOutputs/TwinSafeGroup1.Reset1_45
//     PlcTask Outputs/GVL_IO_SAFETY.bSafetyReset2 <-> StandardOutputs/TwinSafeGroup1.Reset2_46
//     PlcTask Outputs/GVL_IO_SAFETY.bSafetyReset3 <-> StandardOutputs/TwinSafeGroup1.Reset3_83

CONFIGURATION ProgramPLC
    RESOURCE PLC ON TwinCAT3
        TASK PlcTask(INTERVAL := T#3ms, PRIORITY := 20);
        TASK WeightTask(INTERVAL := T#2ms, PRIORITY := 19);
        PROGRAM MAIN WITH PlcTask : MAIN;
        PROGRAM P05_Weight WITH WeightTask : P05_Weight;
    END_RESOURCE
END_CONFIGURATION

// ---- DUTs/AxisControl/ST_AxisControlHoldingBrake.TcDUT
TYPE ST_AxisControlHoldingBrake :
STRUCT
	bReleaseBrake								: BOOL;
	bLockBrake									: BOOL;
END_STRUCT
END_TYPE

// ---- DUTs/AxisControl/ST_AxisControlLS.TcDUT
// modulo (shortest way)/absolute movements
// -- - + ++
// move / pos / velo
// stop / reset
// 
TYPE ST_AxisControlLS :
STRUCT
	bLimitSwitchStateMin						: BOOL;
	bLimitSwitchStateMax						: BOOL;
	bWriteLS									: BOOL;
	bReadLS										: BOOL;
	fLimitSwitchPositionMax						: LREAL;
	fLimitSwitchPositionMin						: LREAL;
END_STRUCT
END_TYPE

// ---- DUTs/AxisControl/ST_AxisControlManual.TcDUT
// modulo (shortest way)/absolute movements
// -- - + ++
// move / pos / velo
// stop / reset
TYPE ST_AxisControlManual :
STRUCT
	bEnable										: BOOL;
	bModulo										: BOOL;
	bSlowForward								: BOOL;
	bSlowBackward								: BOOL;
	bFastForward								: BOOL;
	bFastBackward								: BOOL;
	bStop										: BOOL;
	bReset										: BOOL;
	bExecute									: BOOL;
	fVelocity									: LREAL;
	fPosition									: LREAL;
	fOverride									: LREAL;
END_STRUCT
END_TYPE

